LIN {X -0.031,Y -138.979,Z 1081.101,A 0.000,B 0.000,C 90.000,E1 198.181} C_DIS
LIN {X -0.046,Y -138.332,Z 1081.054,A 0.000,B 0.000,C 90.000,E1 189.782} C_DIS
LIN {X -0.046,Y -139.429,Z 1081.008,A 0.000,B 0.000,C 90.000,E1 181.375} C_DIS
LIN {X 0.007,Y -141.357,Z 1080.971,A 0.000,B 0.000,C 90.000,E1 174.837} C_DIS
LIN {X -0.016,Y -142.711,Z 1080.956,A 0.000,B 0.000,C 90.000,E1 172.064} C_DIS
LIN {X -0.057,Y -145.086,Z 1080.930,A 0.000,B 0.000,C 90.000,E1 167.465} C_DIS
LIN {X -0.062,Y -147.710,Z 1080.910,A 0.000,B 0.000,C 90.000,E1 163.795} C_DIS
LIN {X 0.022,Y -150.365,Z 1080.890,A 0.000,B 0.000,C 90.000,E1 160.115} C_DIS
LIN {X 0.040,Y -153.792,Z 1080.870,A 0.000,B 0.000,C 90.000,E1 156.485} C_DIS
LIN {X -0.040,Y -157.204,Z 1080.849,A 0.000,B 0.000,C 90.000,E1 152.922} C_DIS
LIN {X 0.041,Y -161.367,Z 1080.830,A 0.000,B 0.000,C 90.000,E1 149.331} C_DIS
LIN {X 0.053,Y -165.569,Z 1080.810,A 0.000,B 0.000,C 90.000,E1 145.801} C_DIS
LIN {X -0.064,Y -170.487,Z 1080.791,A 0.000,B 0.000,C 90.000,E1 142.351} C_DIS
LIN {X 0.086,Y -175.368,Z 1080.772,A 0.000,B 0.000,C 90.000,E1 138.852} C_DIS
LIN {X -0.052,Y -180.992,Z 1080.753,A 0.000,B 0.000,C 90.000,E1 135.486} C_DIS
LIN {X 0.073,Y -186.419,Z 1080.734,A 0.000,B 0.000,C 90.000,E1 132.081} C_DIS
LIN {X -0.127,Y -191.046,Z 1080.720,A 0.000,B 0.000,C 90.000,E1 129.644} C_DIS
LIN {X 0.065,Y -196.830,Z 1080.702,A 0.000,B 0.000,C 90.000,E1 126.297} C_DIS
LIN {X -0.010,Y -199.393,Z 1080.695,A 0.000,B 0.000,C 90.000,E1 125.025} C_DIS
LIN {X -0.069,Y -306.720,Z 1080.694,A 0.000,B 0.000,C 90.000,E1 125.025} C_DIS
LIN {X 0.023,Y -308.438,Z 1080.694,A 0.000,B 0.000,C 90.000,E1 124.978} C_DIS
LIN {X -0.026,Y -314.042,Z 1080.693,A 0.000,B 0.000,C 90.000,E1 124.692} C_DIS
LIN {X 0.025,Y -317.211,Z 1080.691,A 0.000,B 0.000,C 90.000,E1 124.358} C_DIS
LIN {X 0.033,Y -319.218,Z 1080.689,A 0.000,B 0.000,C 90.000,E1 124.072} C_DIS
LIN {X 0.038,Y -320.797,Z 1080.688,A 0.000,B 0.000,C 90.000,E1 123.785} C_DIS
LIN {X -0.151,Y -322.205,Z 1080.686,A 0.000,B 0.000,C 90.000,E1 123.499} C_DIS
LIN {X -0.148,Y -333.797,Z 1080.668,A 0.000,B 0.000,C 90.000,E1 120.335} C_DIS
LIN {X 0.027,Y -345.608,Z 1080.653,A 0.000,B 0.000,C 90.000,E1 117.513} C_DIS
LIN {X 0.075,Y -358.869,Z 1080.638,A 0.000,B 0.000,C 90.000,E1 114.771} C_DIS
LIN {X 0.107,Y -371.973,Z 1080.625,A 0.000,B 0.000,C 90.000,E1 112.386} C_DIS
LIN {X 0.047,Y -386.409,Z 1080.612,A 0.000,B 0.000,C 90.000,E1 110.066} C_DIS
LIN {X -0.152,Y -402.280,Z 1080.599,A 0.000,B 0.000,C 90.000,E1 107.819} C_DIS
LIN {X -0.217,Y -419.698,Z 1080.587,A 0.000,B 0.000,C 90.000,E1 105.607} C_DIS
LIN {X 0.053,Y -438.766,Z 1080.575,A 0.000,B 0.000,C 90.000,E1 103.411} C_DIS
LIN {X -0.227,Y -458.853,Z 1080.563,A 0.000,B 0.000,C 90.000,E1 101.422} C_DIS
LIN {X 0.154,Y -466.543,Z 1080.559,A 0.000,B 0.000,C 90.000,E1 100.658} C_DIS
LIN {X 0.100,Y -468.893,Z 1080.558,A 0.000,B 0.000,C 90.000,E1 100.433} C_DIS
LIN {X 0.129,Y -470.675,Z 1080.557,A 0.000,B 0.000,C 90.000,E1 100.197} C_DIS
LIN {X -0.017,Y -472.152,Z 1080.555,A 0.000,B 0.000,C 90.000,E1 99.962} C_DIS
LIN {X -0.166,Y -473.255,Z 1080.554,A 0.000,B 0.000,C 90.000,E1 99.726} C_DIS
LIN {X -0.057,Y -474.562,Z 1080.551,A 0.000,B 0.000,C 90.000,E1 99.208} C_DIS
LIN {X 0.134,Y -474.854,Z 1080.548,A 0.000,B 0.000,C 90.000,E1 98.681} C_DIS
LIN {X -0.211,Y -474.182,Z 1080.546,A 0.000,B 0.000,C 90.000,E1 98.219} C_DIS
LIN {X -0.081,Y -472.439,Z 1080.543,A 0.000,B 0.000,C 90.000,E1 97.701} C_DIS
LIN {X 0.246,Y -471.068,Z 1080.541,A 0.000,B 0.000,C 90.000,E1 97.409} C_DIS
LIN {X 0.119,Y -456.819,Z 1080.530,A 0.000,B 0.000,C 90.000,E1 95.391} C_DIS
LIN {X -0.179,Y -440.793,Z 1080.517,A 0.000,B 0.000,C 90.000,E1 93.094} C_DIS
LIN {X -0.040,Y -426.238,Z 1080.504,A 0.000,B 0.000,C 90.000,E1 90.688} C_DIS
LIN {X 0.135,Y -412.442,Z 1080.490,A 0.000,B 0.000,C 90.000,E1 88.224} C_DIS
LIN {X -0.194,Y -403.581,Z 1080.481,A 0.000,B 0.000,C 90.000,E1 86.617} C_DIS
LIN {X 0.099,Y -396.041,Z 1080.473,A 0.000,B 0.000,C 90.000,E1 85.179} C_DIS
LIN {X -0.069,Y -385.270,Z 1080.462,A 0.000,B 0.000,C 90.000,E1 83.223} C_DIS
LIN {X -0.004,Y -375.970,Z 1080.453,A 0.000,B 0.000,C 90.000,E1 81.489} C_DIS
LIN {X -0.045,Y -367.960,Z 1080.445,A 0.000,B 0.000,C 90.000,E1 80.038} C_DIS
LIN {X -0.168,Y -358.125,Z 1080.435,A 0.000,B 0.000,C 90.000,E1 78.285} C_DIS
LIN {X -0.044,Y -348.134,Z 1080.425,A 0.000,B 0.000,C 90.000,E1 76.464} C_DIS
LIN {X 0.188,Y -334.929,Z 1080.411,A 0.000,B 0.000,C 90.000,E1 73.976} C_DIS
LIN {X -0.184,Y -320.619,Z 1080.396,A 0.000,B 0.000,C 90.000,E1 71.221} C_DIS
LIN {X -0.014,Y -305.773,Z 1080.378,A 0.000,B 0.000,C 90.000,E1 67.975} C_DIS
LIN {X -0.091,Y -294.365,Z 1080.363,A 0.000,B 0.000,C 90.000,E1 65.357} C_DIS
LIN {X -0.072,Y -283.185,Z 1080.348,A 0.000,B 0.000,C 90.000,E1 62.666} C_DIS
LIN {X -0.064,Y -272.260,Z 1080.333,A 0.000,B 0.000,C 90.000,E1 59.921} C_DIS
LIN {X -0.013,Y -260.423,Z 1080.315,A 0.000,B 0.000,C 90.000,E1 56.755} C_DIS
LIN {X -0.074,Y -249.075,Z 1080.297,A 0.000,B 0.000,C 90.000,E1 53.543} C_DIS
LIN {X -0.021,Y -238.335,Z 1080.279,A 0.000,B 0.000,C 90.000,E1 50.231} C_DIS
LIN {X -0.028,Y -228.308,Z 1080.260,A 0.000,B 0.000,C 90.000,E1 46.863} C_DIS
LIN {X 0.095,Y -219.962,Z 1080.243,A 0.000,B 0.000,C 90.000,E1 43.785} C_DIS
LIN {X 0.030,Y -211.982,Z 1080.226,A 0.000,B 0.000,C 90.000,E1 40.701} C_DIS
LIN {X -0.048,Y -204.413,Z 1080.209,A 0.000,B 0.000,C 90.000,E1 37.569} C_DIS
LIN {X 0.085,Y -197.482,Z 1080.191,A 0.000,B 0.000,C 90.000,E1 34.326} C_DIS
LIN {X 0.049,Y -191.144,Z 1080.173,A 0.000,B 0.000,C 90.000,E1 31.082} C_DIS
LIN {X 0.090,Y -185.554,Z 1080.154,A 0.000,B 0.000,C 90.000,E1 27.769} C_DIS
LIN {X -0.022,Y -180.742,Z 1080.136,A 0.000,B 0.000,C 90.000,E1 24.463} C_DIS
LIN {X -0.063,Y -176.577,Z 1080.117,A 0.000,B 0.000,C 90.000,E1 21.099} C_DIS
LIN {X -0.069,Y -173.092,Z 1080.098,A 0.000,B 0.000,C 90.000,E1 17.692} C_DIS
LIN {X 0.045,Y -169.742,Z 1080.074,A 0.000,B 0.000,C 90.000,E1 13.355} C_DIS
LIN {X 0.023,Y -167.058,Z 1080.045,A 0.000,B 0.000,C 90.000,E1 8.163} C_DIS
LIN {X 0.051,Y -167.588,Z 1079.954,A 0.000,B 0.000,C 90.000,E1 351.659} C_DIS
LIN {X -0.059,Y -170.073,Z 1079.930,A 0.000,B 0.000,C 90.000,E1 347.353} C_DIS
LIN {X 0.007,Y -173.624,Z 1079.906,A 0.000,B 0.000,C 90.000,E1 343.015} C_DIS
LIN {X 0.062,Y -178.236,Z 1079.882,A 0.000,B 0.000,C 90.000,E1 338.720} C_DIS
LIN {X -0.018,Y -182.666,Z 1079.863,A 0.000,B 0.000,C 90.000,E1 335.357} C_DIS
LIN {X 0.076,Y -187.791,Z 1079.844,A 0.000,B 0.000,C 90.000,E1 331.975} C_DIS
LIN {X -0.097,Y -192.235,Z 1079.831,A 0.000,B 0.000,C 90.000,E1 329.537} C_DIS
LIN {X 0.048,Y -198.868,Z 1079.812,A 0.000,B 0.000,C 90.000,E1 326.215} C_DIS
LIN {X -0.027,Y -206.227,Z 1079.794,A 0.000,B 0.000,C 90.000,E1 323.004} C_DIS
LIN {X -0.128,Y -215.311,Z 1079.775,A 0.000,B 0.000,C 90.000,E1 319.461} C_DIS
LIN {X 0.000,Y -225.348,Z 1079.755,A 0.000,B 0.000,C 90.000,E1 315.931} C_DIS
LIN {X -0.025,Y -235.355,Z 1079.738,A 0.000,B 0.000,C 90.000,E1 312.894} C_DIS
LIN {X 0.113,Y -243.794,Z 1079.726,A 0.000,B 0.000,C 90.000,E1 310.620} C_DIS
LIN {X -0.065,Y -254.986,Z 1079.712,A 0.000,B 0.000,C 90.000,E1 308.096} C_DIS
LIN {X -0.011,Y -265.577,Z 1079.700,A 0.000,B 0.000,C 90.000,E1 305.931} C_DIS
LIN {X 0.140,Y -282.884,Z 1079.682,A 0.000,B 0.000,C 90.000,E1 302.752} C_DIS
LIN {X -0.038,Y -301.712,Z 1079.665,A 0.000,B 0.000,C 90.000,E1 299.745} C_DIS
LIN {X -0.051,Y -319.749,Z 1079.651,A 0.000,B 0.000,C 90.000,E1 297.129} C_DIS
LIN {X 0.005,Y -331.675,Z 1079.642,A 0.000,B 0.000,C 90.000,E1 295.540} C_DIS
LIN {X -0.092,Y -344.652,Z 1079.633,A 0.000,B 0.000,C 90.000,E1 294.003} C_DIS
LIN {X -0.034,Y -360.721,Z 1079.624,A 0.000,B 0.000,C 90.000,E1 292.280} C_DIS
LIN {X 0.134,Y -379.510,Z 1079.614,A 0.000,B 0.000,C 90.000,E1 290.482} C_DIS
LIN {X -0.097,Y -398.773,Z 1079.605,A 0.000,B 0.000,C 90.000,E1 288.852} C_DIS
LIN {X -0.116,Y -409.487,Z 1079.599,A 0.000,B 0.000,C 90.000,E1 287.928} C_DIS
LIN {X -0.081,Y -419.968,Z 1079.594,A 0.000,B 0.000,C 90.000,E1 286.985} C_DIS
LIN {X -0.117,Y -427.580,Z 1079.590,A 0.000,B 0.000,C 90.000,E1 286.260} C_DIS
LIN {X -0.015,Y -435.113,Z 1079.586,A 0.000,B 0.000,C 90.000,E1 285.481} C_DIS
LIN {X -0.191,Y -442.406,Z 1079.582,A 0.000,B 0.000,C 90.000,E1 284.717} C_DIS
LIN {X 0.146,Y -449.233,Z 1079.577,A 0.000,B 0.000,C 90.000,E1 283.883} C_DIS
LIN {X -0.005,Y -455.567,Z 1079.573,A 0.000,B 0.000,C 90.000,E1 283.119} C_DIS
LIN {X -0.097,Y -461.188,Z 1079.569,A 0.000,B 0.000,C 90.000,E1 282.355} C_DIS
LIN {X -0.149,Y -466.074,Z 1079.564,A 0.000,B 0.000,C 90.000,E1 281.591} C_DIS
LIN {X -0.243,Y -470.161,Z 1079.560,A 0.000,B 0.000,C 90.000,E1 280.838} C_DIS
LIN {X 0.248,Y -473.587,Z 1079.556,A 0.000,B 0.000,C 90.000,E1 280.018} C_DIS
LIN {X -0.110,Y -475.562,Z 1079.553,A 0.000,B 0.000,C 90.000,E1 279.557} C_DIS
LIN {X 0.086,Y -477.292,Z 1079.550,A 0.000,B 0.000,C 90.000,E1 279.029} C_DIS
LIN {X -0.112,Y -480.068,Z 1079.545,A 0.000,B 0.000,C 90.000,E1 278.049} C_DIS
LIN {X 0.208,Y -482.037,Z 1079.539,A 0.000,B 0.000,C 90.000,E1 277.011} C_DIS
LIN {X -0.099,Y -482.717,Z 1079.536,A 0.000,B 0.000,C 90.000,E1 276.549} C_DIS
LIN {X 0.078,Y -483.184,Z 1079.534,A 0.000,B 0.000,C 90.000,E1 276.030} C_DIS
LIN {X -0.223,Y -483.240,Z 1079.531,A 0.000,B 0.000,C 90.000,E1 275.568} C_DIS
LIN {X -0.040,Y -482.989,Z 1079.528,A 0.000,B 0.000,C 90.000,E1 275.049} C_DIS
LIN {X 0.139,Y -482.213,Z 1079.525,A 0.000,B 0.000,C 90.000,E1 274.531} C_DIS
LIN {X -0.165,Y -480.947,Z 1079.522,A 0.000,B 0.000,C 90.000,E1 274.069} C_DIS
LIN {X -0.026,Y -479.128,Z 1079.520,A 0.000,B 0.000,C 90.000,E1 273.555} C_DIS
LIN {X 0.134,Y -476.657,Z 1079.517,A 0.000,B 0.000,C 90.000,E1 273.037} C_DIS
LIN {X -0.223,Y -473.411,Z 1079.514,A 0.000,B 0.000,C 90.000,E1 272.579} C_DIS
LIN {X -0.119,Y -469.277,Z 1079.511,A 0.000,B 0.000,C 90.000,E1 272.064} C_DIS
LIN {X -0.021,Y -464.125,Z 1079.509,A 0.000,B 0.000,C 90.000,E1 271.547} C_DIS
LIN {X -0.149,Y -458.207,Z 1079.506,A 0.000,B 0.000,C 90.000,E1 271.088} C_DIS
LIN {X 0.162,Y -451.915,Z 1079.504,A 0.000,B 0.000,C 90.000,E1 270.630} C_DIS
LIN {X 0.015,Y -445.005,Z 1079.502,A 0.000,B 0.000,C 90.000,E1 270.286} C_DIS
LIN {X -0.052,Y -437.619,Z 1079.500,A 0.000,B 0.000,C 90.000,E1 270.000} C_DIS
LIN {X -0.035,Y -430.037,Z 1079.499,A 0.000,B 0.000,C 90.000,E1 269.771} C_DIS
LIN {X -0.036,Y -422.471,Z 1079.498,A 0.000,B 0.000,C 90.000,E1 269.599} C_DIS
LIN {X -0.167,Y -414.182,Z 1079.497,A 0.000,B 0.000,C 90.000,E1 269.484} C_DIS
LIN {X -0.071,Y -404.523,Z 1079.496,A 0.000,B 0.000,C 90.000,E1 269.370} C_DIS
LIN {X 0.006,Y -396.170,Z 1079.496,A 0.000,B 0.000,C 90.000,E1 269.312} C_DIS
LIN {X -0.059,Y -391.384,Z 1079.496,A 0.000,B 0.000,C 90.000,E1 269.312} C_DIS
LIN {X -0.057,Y -181.388,Z 1079.496,A 0.000,B 0.000,C 90.000,E1 269.312} C_DIS
LIN {X 0.061,Y -180.784,Z 1079.471,A 0.000,B 0.000,C 90.000,E1 264.723} C_DIS
LIN {X -0.045,Y -178.881,Z 1079.443,A 0.000,B 0.000,C 90.000,E1 259.690} C_DIS
LIN {X 0.032,Y -175.923,Z 1079.414,A 0.000,B 0.000,C 90.000,E1 254.574} C_DIS
LIN {X -0.023,Y -175.361,Z 1079.410,A 0.000,B 0.000,C 90.000,E1 253.740} C_DIS
LIN {X 0.036,Y -172.140,Z 1079.386,A 0.000,B 0.000,C 90.000,E1 249.444} C_DIS
LIN {X 0.013,Y -171.604,Z 1079.381,A 0.000,B 0.000,C 90.000,E1 248.592} C_DIS
LIN {X 0.002,Y -167.826,Z 1079.357,A 0.000,B 0.000,C 90.000,E1 244.280} C_DIS
LIN {X 0.019,Y -166.551,Z 1079.347,A 0.000,B 0.000,C 90.000,E1 242.538} C_DIS
LIN {X -0.070,Y -162.547,Z 1079.323,A 0.000,B 0.000,C 90.000,E1 238.201} C_DIS
LIN {X -0.010,Y -161.224,Z 1079.313,A 0.000,B 0.000,C 90.000,E1 236.421} C_DIS
LIN {X 0.025,Y -157.230,Z 1079.289,A 0.000,B 0.000,C 90.000,E1 231.984} C_DIS
LIN {X 0.048,Y -155.956,Z 1079.279,A 0.000,B 0.000,C 90.000,E1 230.194} C_DIS
LIN {X 0.006,Y -152.209,Z 1079.254,A 0.000,B 0.000,C 90.000,E1 225.729} C_DIS
LIN {X 0.028,Y -150.454,Z 1079.239,A 0.000,B 0.000,C 90.000,E1 223.014} C_DIS
LIN {X 0.054,Y -147.180,Z 1079.214,A 0.000,B 0.000,C 90.000,E1 218.463} C_DIS
LIN {X 0.020,Y -145.196,Z 1079.193,A 0.000,B 0.000,C 90.000,E1 214.818} C_DIS
LIN {X 0.054,Y -142.336,Z 1079.163,A 0.000,B 0.000,C 90.000,E1 209.283} C_DIS
LIN {X -0.016,Y -141.725,Z 1079.153,A 0.000,B 0.000,C 90.000,E1 207.462} C_DIS
LIN {X -0.034,Y -139.478,Z 1079.116,A 0.000,B 0.000,C 90.000,E1 200.972} C_DIS
LIN {X -0.045,Y -138.978,Z 1079.101,A 0.000,B 0.000,C 90.000,E1 198.181} C_DIS
LIN {X 0.076,Y -138.332,Z 1079.054,A 0.000,B 0.000,C 90.000,E1 189.726} C_DIS
LIN {X -0.059,Y -139.431,Z 1079.007,A 0.000,B 0.000,C 90.000,E1 181.375} C_DIS
LIN {X 0.020,Y -140.956,Z 1078.976,A 0.000,B 0.000,C 90.000,E1 175.755} C_DIS
LIN {X -0.030,Y -142.713,Z 1078.956,A 0.000,B 0.000,C 90.000,E1 172.064} C_DIS
LIN {X 0.070,Y -145.089,Z 1078.930,A 0.000,B 0.000,C 90.000,E1 167.409} C_DIS
LIN {X 0.065,Y -147.713,Z 1078.910,A 0.000,B 0.000,C 90.000,E1 163.740} C_DIS
LIN {X 0.007,Y -150.370,Z 1078.890,A 0.000,B 0.000,C 90.000,E1 160.115} C_DIS
LIN {X 0.025,Y -153.798,Z 1078.869,A 0.000,B 0.000,C 90.000,E1 156.485} C_DIS
LIN {X 0.085,Y -157.210,Z 1078.849,A 0.000,B 0.000,C 90.000,E1 152.871} C_DIS
LIN {X 0.026,Y -161.373,Z 1078.830,A 0.000,B 0.000,C 90.000,E1 149.331} C_DIS
LIN {X 0.038,Y -165.576,Z 1078.810,A 0.000,B 0.000,C 90.000,E1 145.801} C_DIS
LIN {X 0.024,Y -170.496,Z 1078.791,A 0.000,B 0.000,C 90.000,E1 142.316} C_DIS
LIN {X 0.069,Y -175.376,Z 1078.771,A 0.000,B 0.000,C 90.000,E1 138.852} C_DIS
LIN {X -0.068,Y -181.000,Z 1078.753,A 0.000,B 0.000,C 90.000,E1 135.486} C_DIS
LIN {X 0.056,Y -186.428,Z 1078.734,A 0.000,B 0.000,C 90.000,E1 132.081} C_DIS
LIN {X 0.125,Y -191.054,Z 1078.720,A 0.000,B 0.000,C 90.000,E1 129.564} C_DIS
LIN {X 0.048,Y -196.839,Z 1078.702,A 0.000,B 0.000,C 90.000,E1 126.297} C_DIS
LIN {X 0.133,Y -199.309,Z 1078.695,A 0.000,B 0.000,C 90.000,E1 125.025} C_DIS
LIN {X 0.145,Y -306.793,Z 1078.695,A 0.000,B 0.000,C 90.000,E1 125.025} C_DIS
LIN {X -0.037,Y -308.518,Z 1078.695,A 0.000,B 0.000,C 90.000,E1 125.025} C_DIS
LIN {X 0.172,Y -312.221,Z 1078.694,A 0.000,B 0.000,C 90.000,E1 124.818} C_DIS
LIN {X -0.053,Y -314.434,Z 1078.693,A 0.000,B 0.000,C 90.000,E1 124.692} C_DIS
LIN {X -0.074,Y -318.322,Z 1078.690,A 0.000,B 0.000,C 90.000,E1 124.246} C_DIS
LIN {X 0.049,Y -320.192,Z 1078.688,A 0.000,B 0.000,C 90.000,E1 123.913} C_DIS
LIN {X -0.094,Y -321.659,Z 1078.687,A 0.000,B 0.000,C 90.000,E1 123.627} C_DIS
LIN {X 0.140,Y -335.736,Z 1078.666,A 0.000,B 0.000,C 90.000,E1 119.795} C_DIS
LIN {X -0.090,Y -347.789,Z 1078.650,A 0.000,B 0.000,C 90.000,E1 117.052} C_DIS
LIN {X -0.146,Y -361.319,Z 1078.635,A 0.000,B 0.000,C 90.000,E1 114.335} C_DIS
LIN {X -0.060,Y -374.676,Z 1078.622,A 0.000,B 0.000,C 90.000,E1 111.950} C_DIS
LIN {X -0.061,Y -389.386,Z 1078.609,A 0.000,B 0.000,C 90.000,E1 109.631} C_DIS
LIN {X 0.065,Y -405.552,Z 1078.596,A 0.000,B 0.000,C 90.000,E1 107.347} C_DIS
LIN {X 0.097,Y -423.289,Z 1078.584,A 0.000,B 0.000,C 90.000,E1 105.134} C_DIS
LIN {X -0.023,Y -442.658,Z 1078.572,A 0.000,B 0.000,C 90.000,E1 103.008} C_DIS
LIN {X 0.062,Y -462.856,Z 1078.561,A 0.000,B 0.000,C 90.000,E1 101.007} C_DIS
LIN {X -0.023,Y -467.950,Z 1078.559,A 0.000,B 0.000,C 90.000,E1 100.546} C_DIS
LIN {X -0.030,Y -469.985,Z 1078.557,A 0.000,B 0.000,C 90.000,E1 100.310} C_DIS
LIN {X -0.038,Y -471.530,Z 1078.556,A 0.000,B 0.000,C 90.000,E1 100.074} C_DIS
LIN {X 0.201,Y -472.784,Z 1078.555,A 0.000,B 0.000,C 90.000,E1 99.792} C_DIS
LIN {X 0.056,Y -473.704,Z 1078.553,A 0.000,B 0.000,C 90.000,E1 99.557} C_DIS
LIN {X 0.246,Y -474.711,Z 1078.550,A 0.000,B 0.000,C 90.000,E1 99.029} C_DIS
LIN {X -0.103,Y -474.732,Z 1078.547,A 0.000,B 0.000,C 90.000,E1 98.568} C_DIS
LIN {X 0.025,Y -473.777,Z 1078.545,A 0.000,B 0.000,C 90.000,E1 98.049} C_DIS
LIN {X 0.154,Y -471.684,Z 1078.542,A 0.000,B 0.000,C 90.000,E1 97.530} C_DIS
LIN {X -0.187,Y -468.228,Z 1078.539,A 0.000,B 0.000,C 90.000,E1 97.068} C_DIS
LIN {X -0.124,Y -455.799,Z 1078.529,A 0.000,B 0.000,C 90.000,E1 95.277} C_DIS
LIN {X -0.205,Y -441.518,Z 1078.518,A 0.000,B 0.000,C 90.000,E1 93.212} C_DIS
LIN {X 0.113,Y -425.345,Z 1078.503,A 0.000,B 0.000,C 90.000,E1 90.516} C_DIS
LIN {X 0.028,Y -408.666,Z 1078.486,A 0.000,B 0.000,C 90.000,E1 87.535} C_DIS
LIN {X 0.044,Y -399.759,Z 1078.477,A 0.000,B 0.000,C 90.000,E1 85.869} C_DIS
LIN {X -0.048,Y -389.033,Z 1078.466,A 0.000,B 0.000,C 90.000,E1 83.913} C_DIS
LIN {X 0.063,Y -378.216,Z 1078.455,A 0.000,B 0.000,C 90.000,E1 81.894} C_DIS
LIN {X 0.053,Y -368.646,Z 1078.445,A 0.000,B 0.000,C 90.000,E1 80.151} C_DIS
LIN {X -0.129,Y -358.801,Z 1078.436,A 0.000,B 0.000,C 90.000,E1 78.409} C_DIS
LIN {X 0.002,Y -348.832,Z 1078.426,A 0.000,B 0.000,C 90.000,E1 76.589} C_DIS
LIN {X 0.018,Y -337.247,Z 1078.414,A 0.000,B 0.000,C 90.000,E1 74.448} C_DIS
LIN {X 0.027,Y -322.815,Z 1078.398,A 0.000,B 0.000,C 90.000,E1 71.638} C_DIS
LIN {X -0.139,Y -307.817,Z 1078.380,A 0.000,B 0.000,C 90.000,E1 68.465} C_DIS
LIN {X 0.114,Y -296.351,Z 1078.366,A 0.000,B 0.000,C 90.000,E1 65.793} C_DIS
LIN {X 0.069,Y -286.517,Z 1078.353,A 0.000,B 0.000,C 90.000,E1 63.461} C_DIS
LIN {X 0.145,Y -275.497,Z 1078.338,A 0.000,B 0.000,C 90.000,E1 60.717} C_DIS
LIN {X -0.143,Y -264.801,Z 1078.322,A 0.000,B 0.000,C 90.000,E1 57.995} C_DIS
LIN {X 0.094,Y -254.490,Z 1078.306,A 0.000,B 0.000,C 90.000,E1 55.102} C_DIS
LIN {X 0.148,Y -244.623,Z 1078.290,A 0.000,B 0.000,C 90.000,E1 52.190} C_DIS
LIN {X -0.145,Y -234.131,Z 1078.272,A 0.000,B 0.000,C 90.000,E1 48.933} C_DIS
LIN {X -0.041,Y -225.430,Z 1078.255,A 0.000,B 0.000,C 90.000,E1 45.891} C_DIS
LIN {X 0.010,Y -217.158,Z 1078.238,A 0.000,B 0.000,C 90.000,E1 42.813} C_DIS
LIN {X -0.103,Y -209.272,Z 1078.221,A 0.000,B 0.000,C 90.000,E1 39.725} C_DIS
LIN {X 0.075,Y -201.926,Z 1078.203,A 0.000,B 0.000,C 90.000,E1 36.503} C_DIS
LIN {X 0.032,Y -195.149,Z 1078.185,A 0.000,B 0.000,C 90.000,E1 33.293} C_DIS
LIN {X 0.102,Y -189.040,Z 1078.167,A 0.000,B 0.000,C 90.000,E1 30.001} C_DIS
LIN {X -0.089,Y -183.713,Z 1078.148,A 0.000,B 0.000,C 90.000,E1 26.744} C_DIS
LIN {X -0.078,Y -179.114,Z 1078.130,A 0.000,B 0.000,C 90.000,E1 23.387} C_DIS
LIN {X -0.063,Y -175.159,Z 1078.111,A 0.000,B 0.000,C 90.000,E1 19.993} C_DIS
LIN {X 0.002,Y -171.899,Z 1078.092,A 0.000,B 0.000,C 90.000,E1 16.551} C_DIS
LIN {X -0.005,Y -168.836,Z 1078.068,A 0.000,B 0.000,C 90.000,E1 12.243} C_DIS
LIN {X 0.046,Y -166.198,Z 1078.034,A 0.000,B 0.000,C 90.000,E1 6.144} C_DIS
LIN {X 0.029,Y -167.013,Z 1077.959,A 0.000,B 0.000,C 90.000,E1 352.534} C_DIS
LIN {X -0.077,Y -169.876,Z 1077.930,A 0.000,B 0.000,C 90.000,E1 347.353} C_DIS
LIN {X -0.016,Y -173.445,Z 1077.906,A 0.000,B 0.000,C 90.000,E1 343.015} C_DIS
LIN {X 0.034,Y -177.040,Z 1077.887,A 0.000,B 0.000,C 90.000,E1 339.571} C_DIS
LIN {X 0.024,Y -181.331,Z 1077.868,A 0.000,B 0.000,C 90.000,E1 336.177} C_DIS
LIN {X 0.001,Y -186.257,Z 1077.849,A 0.000,B 0.000,C 90.000,E1 332.820} C_DIS
LIN {X -0.035,Y -190.532,Z 1077.835,A 0.000,B 0.000,C 90.000,E1 330.333} C_DIS
LIN {X -0.038,Y -196.978,Z 1077.817,A 0.000,B 0.000,C 90.000,E1 327.041} C_DIS
LIN {X 0.005,Y -204.202,Z 1077.799,A 0.000,B 0.000,C 90.000,E1 323.783} C_DIS
LIN {X -0.019,Y -212.093,Z 1077.781,A 0.000,B 0.000,C 90.000,E1 320.598} C_DIS
LIN {X -0.044,Y -220.675,Z 1077.764,A 0.000,B 0.000,C 90.000,E1 317.472} C_DIS
LIN {X 0.138,Y -230.094,Z 1077.747,A 0.000,B 0.000,C 90.000,E1 314.352} C_DIS
LIN {X -0.044,Y -239.333,Z 1077.732,A 0.000,B 0.000,C 90.000,E1 311.757} C_DIS
LIN {X 0.020,Y -248.271,Z 1077.720,A 0.000,B 0.000,C 90.000,E1 309.519} C_DIS
LIN {X -0.095,Y -258.244,Z 1077.707,A 0.000,B 0.000,C 90.000,E1 307.363} C_DIS
LIN {X 0.066,Y -273.015,Z 1077.692,A 0.000,B 0.000,C 90.000,E1 304.485} C_DIS
LIN {X 0.052,Y -291.007,Z 1077.674,A 0.000,B 0.000,C 90.000,E1 301.386} C_DIS
LIN {X -0.089,Y -308.291,Z 1077.660,A 0.000,B 0.000,C 90.000,E1 298.743} C_DIS
LIN {X -0.102,Y -329.252,Z 1077.644,A 0.000,B 0.000,C 90.000,E1 295.848} C_DIS
LIN {X 0.056,Y -342.075,Z 1077.635,A 0.000,B 0.000,C 90.000,E1 294.259} C_DIS
LIN {X 0.042,Y -355.244,Z 1077.627,A 0.000,B 0.000,C 90.000,E1 292.823} C_DIS
LIN {X -0.032,Y -374.367,Z 1077.616,A 0.000,B 0.000,C 90.000,E1 290.972} C_DIS
LIN {X 0.012,Y -393.690,Z 1077.607,A 0.000,B 0.000,C 90.000,E1 289.268} C_DIS
LIN {X -0.117,Y -407.467,Z 1077.600,A 0.000,B 0.000,C 90.000,E1 288.109} C_DIS
LIN {X 0.005,Y -418.077,Z 1077.595,A 0.000,B 0.000,C 90.000,E1 287.149} C_DIS
LIN {X -0.125,Y -425.791,Z 1077.591,A 0.000,B 0.000,C 90.000,E1 286.441} C_DIS
LIN {X 0.085,Y -433.260,Z 1077.587,A 0.000,B 0.000,C 90.000,E1 285.662} C_DIS
LIN {X 0.000,Y -440.537,Z 1077.583,A 0.000,B 0.000,C 90.000,E1 284.898} C_DIS
LIN {X -0.049,Y -447.485,Z 1077.578,A 0.000,B 0.000,C 90.000,E1 284.120} C_DIS
LIN {X -0.171,Y -453.916,Z 1077.574,A 0.000,B 0.000,C 90.000,E1 283.355} C_DIS
LIN {X 0.165,Y -459.735,Z 1077.570,A 0.000,B 0.000,C 90.000,E1 282.535} C_DIS
LIN {X 0.112,Y -464.865,Z 1077.565,A 0.000,B 0.000,C 90.000,E1 281.771} C_DIS
LIN {X 0.094,Y -469.138,Z 1077.561,A 0.000,B 0.000,C 90.000,E1 281.007} C_DIS
LIN {X 0.031,Y -472.754,Z 1077.557,A 0.000,B 0.000,C 90.000,E1 280.254} C_DIS
LIN {X -0.001,Y -475.834,Z 1077.553,A 0.000,B 0.000,C 90.000,E1 279.500} C_DIS
LIN {X 0.196,Y -477.551,Z 1077.550,A 0.000,B 0.000,C 90.000,E1 278.973} C_DIS
LIN {X -0.142,Y -479.042,Z 1077.547,A 0.000,B 0.000,C 90.000,E1 278.511} C_DIS
LIN {X 0.004,Y -480.332,Z 1077.544,A 0.000,B 0.000,C 90.000,E1 277.992} C_DIS
LIN {X -0.091,Y -482.325,Z 1077.539,A 0.000,B 0.000,C 90.000,E1 277.004} C_DIS
LIN {X 0.078,Y -483.018,Z 1077.536,A 0.000,B 0.000,C 90.000,E1 276.486} C_DIS
LIN {X 0.254,Y -483.442,Z 1077.533,A 0.000,B 0.000,C 90.000,E1 275.967} C_DIS
LIN {X -0.096,Y -483.538,Z 1077.531,A 0.000,B 0.000,C 90.000,E1 275.511} C_DIS
LIN {X 0.088,Y -483.223,Z 1077.528,A 0.000,B 0.000,C 90.000,E1 274.992} C_DIS
LIN {X -0.211,Y -482.431,Z 1077.525,A 0.000,B 0.000,C 90.000,E1 274.531} C_DIS
LIN {X -0.033,Y -481.125,Z 1077.522,A 0.000,B 0.000,C 90.000,E1 274.012} C_DIS
LIN {X 0.106,Y -479.277,Z 1077.520,A 0.000,B 0.000,C 90.000,E1 273.498} C_DIS
LIN {X -0.209,Y -476.758,Z 1077.517,A 0.000,B 0.000,C 90.000,E1 273.037} C_DIS
LIN {X -0.090,Y -473.440,Z 1077.514,A 0.000,B 0.000,C 90.000,E1 272.522} C_DIS
LIN {X 0.014,Y -469.253,Z 1077.511,A 0.000,B 0.000,C 90.000,E1 272.007} C_DIS
LIN {X -0.163,Y -466.788,Z 1077.510,A 0.000,B 0.000,C 90.000,E1 271.776} C_DIS
LIN {X 0.072,Y -461.196,Z 1077.507,A 0.000,B 0.000,C 90.000,E1 271.260} C_DIS
LIN {X 0.189,Y -455.133,Z 1077.505,A 0.000,B 0.000,C 90.000,E1 270.802} C_DIS
LIN {X -0.111,Y -451.816,Z 1077.503,A 0.000,B 0.000,C 90.000,E1 270.630} C_DIS
LIN {X 0.195,Y -444.754,Z 1077.501,A 0.000,B 0.000,C 90.000,E1 270.229} C_DIS
LIN {X -0.030,Y -441.441,Z 1077.501,A 0.000,B 0.000,C 90.000,E1 270.115} C_DIS
LIN {X 0.213,Y -434.099,Z 1077.499,A 0.000,B 0.000,C 90.000,E1 269.828} C_DIS
LIN {X 0.027,Y -426.617,Z 1077.498,A 0.000,B 0.000,C 90.000,E1 269.656} C_DIS
LIN {X 0.183,Y -418.588,Z 1077.497,A 0.000,B 0.000,C 90.000,E1 269.484} C_DIS
LIN {X 0.189,Y -409.875,Z 1077.497,A 0.000,B 0.000,C 90.000,E1 269.370} C_DIS
LIN {X -0.076,Y -396.410,Z 1077.496,A 0.000,B 0.000,C 90.000,E1 269.312} C_DIS
LIN {X -0.139,Y -391.628,Z 1077.496,A 0.000,B 0.000,C 90.000,E1 269.312} C_DIS
LIN {X 0.088,Y -181.384,Z 1077.496,A 0.000,B 0.000,C 90.000,E1 269.255} C_DIS
LIN {X 0.024,Y -180.779,Z 1077.471,A 0.000,B 0.000,C 90.000,E1 264.723} C_DIS
LIN {X -0.081,Y -178.876,Z 1077.443,A 0.000,B 0.000,C 90.000,E1 259.690} C_DIS
LIN {X -0.005,Y -175.919,Z 1077.414,A 0.000,B 0.000,C 90.000,E1 254.574} C_DIS
LIN {X 0.052,Y -174.614,Z 1077.405,A 0.000,B 0.000,C 90.000,E1 252.851} C_DIS
LIN {X -0.023,Y -171.594,Z 1077.381,A 0.000,B 0.000,C 90.000,E1 248.592} C_DIS
LIN {X -0.033,Y -167.817,Z 1077.357,A 0.000,B 0.000,C 90.000,E1 244.280} C_DIS
LIN {X -0.016,Y -166.540,Z 1077.347,A 0.000,B 0.000,C 90.000,E1 242.538} C_DIS
LIN {X -0.106,Y -162.537,Z 1077.323,A 0.000,B 0.000,C 90.000,E1 238.201} C_DIS
LIN {X -0.045,Y -161.213,Z 1077.313,A 0.000,B 0.000,C 90.000,E1 236.421} C_DIS
LIN {X -0.009,Y -157.221,Z 1077.289,A 0.000,B 0.000,C 90.000,E1 231.984} C_DIS
LIN {X 0.014,Y -155.947,Z 1077.279,A 0.000,B 0.000,C 90.000,E1 230.194} C_DIS
LIN {X -0.027,Y -152.200,Z 1077.254,A 0.000,B 0.000,C 90.000,E1 225.729} C_DIS
LIN {X -0.006,Y -150.446,Z 1077.239,A 0.000,B 0.000,C 90.000,E1 223.014} C_DIS
LIN {X 0.021,Y -147.172,Z 1077.214,A 0.000,B 0.000,C 90.000,E1 218.463} C_DIS
LIN {X -0.012,Y -145.188,Z 1077.193,A 0.000,B 0.000,C 90.000,E1 214.818} C_DIS
LIN {X 0.023,Y -142.331,Z 1077.163,A 0.000,B 0.000,C 90.000,E1 209.283} C_DIS
LIN {X -0.047,Y -141.720,Z 1077.152,A 0.000,B 0.000,C 90.000,E1 207.462} C_DIS
LIN {X 0.065,Y -139.476,Z 1077.116,A 0.000,B 0.000,C 90.000,E1 200.918} C_DIS
LIN {X -0.076,Y -138.974,Z 1077.101,A 0.000,B 0.000,C 90.000,E1 198.181} C_DIS
LIN {X 0.045,Y -138.331,Z 1077.054,A 0.000,B 0.000,C 90.000,E1 189.726} C_DIS
LIN {X 0.048,Y -139.434,Z 1077.007,A 0.000,B 0.000,C 90.000,E1 181.318} C_DIS
LIN {X -0.012,Y -140.962,Z 1076.976,A 0.000,B 0.000,C 90.000,E1 175.755} C_DIS
LIN {X -0.062,Y -142.717,Z 1076.956,A 0.000,B 0.000,C 90.000,E1 172.064} C_DIS
LIN {X 0.038,Y -145.097,Z 1076.930,A 0.000,B 0.000,C 90.000,E1 167.409} C_DIS
LIN {X 0.032,Y -147.722,Z 1076.910,A 0.000,B 0.000,C 90.000,E1 163.740} C_DIS
LIN {X -0.027,Y -150.380,Z 1076.890,A 0.000,B 0.000,C 90.000,E1 160.115} C_DIS
LIN {X -0.009,Y -153.811,Z 1076.869,A 0.000,B 0.000,C 90.000,E1 156.485} C_DIS
LIN {X 0.051,Y -157.223,Z 1076.849,A 0.000,B 0.000,C 90.000,E1 152.871} C_DIS
LIN {X -0.008,Y -161.389,Z 1076.830,A 0.000,B 0.000,C 90.000,E1 149.331} C_DIS
LIN {X 0.002,Y -165.591,Z 1076.810,A 0.000,B 0.000,C 90.000,E1 145.801} C_DIS
LIN {X -0.011,Y -170.514,Z 1076.791,A 0.000,B 0.000,C 90.000,E1 142.316} C_DIS
LIN {X 0.033,Y -175.394,Z 1076.771,A 0.000,B 0.000,C 90.000,E1 138.852} C_DIS
LIN {X -0.105,Y -181.018,Z 1076.753,A 0.000,B 0.000,C 90.000,E1 135.486} C_DIS
LIN {X 0.018,Y -186.448,Z 1076.734,A 0.000,B 0.000,C 90.000,E1 132.081} C_DIS
LIN {X 0.087,Y -191.074,Z 1076.720,A 0.000,B 0.000,C 90.000,E1 129.564} C_DIS
LIN {X 0.009,Y -196.861,Z 1076.702,A 0.000,B 0.000,C 90.000,E1 126.297} C_DIS
LIN {X 0.024,Y -199.211,Z 1076.695,A 0.000,B 0.000,C 90.000,E1 125.105} C_DIS
LIN {X -0.005,Y -305.919,Z 1076.695,A 0.000,B 0.000,C 90.000,E1 125.105} C_DIS
LIN {X -0.060,Y -312.160,Z 1076.694,A 0.000,B 0.000,C 90.000,E1 124.898} C_DIS
LIN {X -0.115,Y -314.857,Z 1076.693,A 0.000,B 0.000,C 90.000,E1 124.692} C_DIS
LIN {X 0.008,Y -318.653,Z 1076.690,A 0.000,B 0.000,C 90.000,E1 124.199} C_DIS
LIN {X 0.072,Y -320.467,Z 1076.688,A 0.000,B 0.000,C 90.000,E1 123.865} C_DIS
LIN {X -0.131,Y -321.883,Z 1076.686,A 0.000,B 0.000,C 90.000,E1 123.579} C_DIS
LIN {X -0.005,Y -334.672,Z 1076.667,A 0.000,B 0.000,C 90.000,E1 120.079} C_DIS
LIN {X -0.104,Y -346.597,Z 1076.652,A 0.000,B 0.000,C 90.000,E1 117.308} C_DIS
LIN {X -0.041,Y -359.983,Z 1076.636,A 0.000,B 0.000,C 90.000,E1 114.567} C_DIS
LIN {X -0.136,Y -373.205,Z 1076.623,A 0.000,B 0.000,C 90.000,E1 112.206} C_DIS
LIN {X -0.038,Y -387.768,Z 1076.610,A 0.000,B 0.000,C 90.000,E1 109.866} C_DIS
LIN {X 0.041,Y -403.777,Z 1076.598,A 0.000,B 0.000,C 90.000,E1 107.583} C_DIS
LIN {X 0.024,Y -421.344,Z 1076.585,A 0.000,B 0.000,C 90.000,E1 105.371} C_DIS
LIN {X -0.172,Y -440.562,Z 1076.573,A 0.000,B 0.000,C 90.000,E1 103.244} C_DIS
LIN {X 0.218,Y -460.702,Z 1076.562,A 0.000,B 0.000,C 90.000,E1 101.186} C_DIS
LIN {X 0.106,Y -468.312,Z 1076.558,A 0.000,B 0.000,C 90.000,E1 100.489} C_DIS
LIN {X 0.076,Y -470.269,Z 1076.557,A 0.000,B 0.000,C 90.000,E1 100.254} C_DIS
LIN {X 0.044,Y -471.755,Z 1076.556,A 0.000,B 0.000,C 90.000,E1 100.018} C_DIS
LIN {X -0.181,Y -472.942,Z 1076.554,A 0.000,B 0.000,C 90.000,E1 99.792} C_DIS
LIN {X 0.141,Y -473.807,Z 1076.553,A 0.000,B 0.000,C 90.000,E1 99.500} C_DIS
LIN {X -0.136,Y -474.718,Z 1076.550,A 0.000,B 0.000,C 90.000,E1 99.029} C_DIS
LIN {X -0.015,Y -474.652,Z 1076.547,A 0.000,B 0.000,C 90.000,E1 98.511} C_DIS
LIN {X 0.113,Y -473.601,Z 1076.544,A 0.000,B 0.000,C 90.000,E1 97.992} C_DIS
LIN {X -0.024,Y -472.661,Z 1076.543,A 0.000,B 0.000,C 90.000,E1 97.757} C_DIS
LIN {X -0.225,Y -471.387,Z 1076.542,A 0.000,B 0.000,C 90.000,E1 97.530} C_DIS
LIN {X 0.127,Y -460.743,Z 1076.533,A 0.000,B 0.000,C 90.000,E1 95.967} C_DIS
LIN {X -0.026,Y -451.759,Z 1076.526,A 0.000,B 0.000,C 90.000,E1 94.702} C_DIS
LIN {X 0.066,Y -439.527,Z 1076.516,A 0.000,B 0.000,C 90.000,E1 92.865} C_DIS
LIN {X -0.126,Y -423.466,Z 1076.501,A 0.000,B 0.000,C 90.000,E1 90.229} C_DIS
LIN {X 0.141,Y -406.936,Z 1076.484,A 0.000,B 0.000,C 90.000,E1 87.192} C_DIS
LIN {X 0.121,Y -397.958,Z 1076.475,A 0.000,B 0.000,C 90.000,E1 85.527} C_DIS
LIN {X -0.014,Y -387.214,Z 1076.464,A 0.000,B 0.000,C 90.000,E1 83.571} C_DIS
LIN {X 0.083,Y -377.917,Z 1076.455,A 0.000,B 0.000,C 90.000,E1 81.837} C_DIS
LIN {X 0.066,Y -368.343,Z 1076.445,A 0.000,B 0.000,C 90.000,E1 80.095} C_DIS
LIN {X -0.052,Y -358.454,Z 1076.435,A 0.000,B 0.000,C 90.000,E1 78.342} C_DIS
LIN {X 0.008,Y -346.825,Z 1076.423,A 0.000,B 0.000,C 90.000,E1 76.228} C_DIS
LIN {X -0.115,Y -333.636,Z 1076.410,A 0.000,B 0.000,C 90.000,E1 73.795} C_DIS
LIN {X 0.140,Y -317.857,Z 1076.392,A 0.000,B 0.000,C 90.000,E1 70.604} C_DIS
LIN {X 0.013,Y -306.048,Z 1076.378,A 0.000,B 0.000,C 90.000,E1 68.050} C_DIS
LIN {X 0.059,Y -294.643,Z 1076.363,A 0.000,B 0.000,C 90.000,E1 65.409} C_DIS
LIN {X -0.047,Y -283.421,Z 1076.349,A 0.000,B 0.000,C 90.000,E1 62.743} C_DIS
LIN {X -0.040,Y -272.500,Z 1076.333,A 0.000,B 0.000,C 90.000,E1 59.999} C_DIS
LIN {X 0.017,Y -260.574,Z 1076.316,A 0.000,B 0.000,C 90.000,E1 56.834} C_DIS
LIN {X -0.050,Y -249.171,Z 1076.298,A 0.000,B 0.000,C 90.000,E1 53.623} C_DIS
LIN {X 0.006,Y -238.347,Z 1076.280,A 0.000,B 0.000,C 90.000,E1 50.312} C_DIS
LIN {X 0.043,Y -229.324,Z 1076.263,A 0.000,B 0.000,C 90.000,E1 47.310} C_DIS
LIN {X 0.030,Y -220.867,Z 1076.246,A 0.000,B 0.000,C 90.000,E1 44.271} C_DIS
LIN {X 0.131,Y -212.791,Z 1076.229,A 0.000,B 0.000,C 90.000,E1 41.148} C_DIS
LIN {X 0.072,Y -205.120,Z 1076.211,A 0.000,B 0.000,C 90.000,E1 38.016} C_DIS
LIN {X 0.059,Y -198.056,Z 1076.193,A 0.000,B 0.000,C 90.000,E1 34.818} C_DIS
LIN {X -0.022,Y -191.638,Z 1076.175,A 0.000,B 0.000,C 90.000,E1 31.592} C_DIS
LIN {X 0.027,Y -185.948,Z 1076.157,A 0.000,B 0.000,C 90.000,E1 28.281} C_DIS
LIN {X 0.002,Y -181.008,Z 1076.139,A 0.000,B 0.000,C 90.000,E1 24.951} C_DIS
LIN {X -0.038,Y -176.749,Z 1076.120,A 0.000,B 0.000,C 90.000,E1 21.589} C_DIS
LIN {X -0.039,Y -173.150,Z 1076.101,A 0.000,B 0.000,C 90.000,E1 18.181} C_DIS
LIN {X -0.041,Y -169.679,Z 1076.077,A 0.000,B 0.000,C 90.000,E1 13.883} C_DIS
LIN {X -0.037,Y -166.863,Z 1076.048,A 0.000,B 0.000,C 90.000,E1 8.681} C_DIS
LIN {X 0.017,Y -167.606,Z 1075.949,A 0.000,B 0.000,C 90.000,E1 350.792} C_DIS
LIN {X -0.027,Y -170.316,Z 1075.925,A 0.000,B 0.000,C 90.000,E1 346.464} C_DIS
LIN {X 0.049,Y -174.091,Z 1075.901,A 0.000,B 0.000,C 90.000,E1 342.127} C_DIS
LIN {X 0.003,Y -177.870,Z 1075.882,A 0.000,B 0.000,C 90.000,E1 338.720} C_DIS
LIN {X -0.087,Y -182.327,Z 1075.863,A 0.000,B 0.000,C 90.000,E1 335.357} C_DIS
LIN {X -0.004,Y -187.479,Z 1075.844,A 0.000,B 0.000,C 90.000,E1 331.975} C_DIS
LIN {X -0.018,Y -193.533,Z 1075.826,A 0.000,B 0.000,C 90.000,E1 328.663} C_DIS
LIN {X -0.005,Y -200.393,Z 1075.808,A 0.000,B 0.000,C 90.000,E1 325.388} C_DIS
LIN {X -0.088,Y -207.938,Z 1075.790,A 0.000,B 0.000,C 90.000,E1 322.190} C_DIS
LIN {X 0.015,Y -217.277,Z 1075.770,A 0.000,B 0.000,C 90.000,E1 318.609} C_DIS
LIN {X 0.118,Y -226.338,Z 1075.753,A 0.000,B 0.000,C 90.000,E1 315.486} C_DIS
LIN {X 0.010,Y -235.122,Z 1075.738,A 0.000,B 0.000,C 90.000,E1 312.852} C_DIS
LIN {X -0.033,Y -243.545,Z 1075.726,A 0.000,B 0.000,C 90.000,E1 310.620} C_DIS
LIN {X 0.115,Y -252.973,Z 1075.713,A 0.000,B 0.000,C 90.000,E1 308.382} C_DIS
LIN {X -0.020,Y -263.510,Z 1075.701,A 0.000,B 0.000,C 90.000,E1 306.251} C_DIS
LIN {X 0.008,Y -280.781,Z 1075.684,A 0.000,B 0.000,C 90.000,E1 303.086} C_DIS
LIN {X 0.160,Y -299.508,Z 1075.667,A 0.000,B 0.000,C 90.000,E1 300.001} C_DIS
LIN {X 0.016,Y -319.732,Z 1075.650,A 0.000,B 0.000,C 90.000,E1 297.078} C_DIS
LIN {X -0.039,Y -334.105,Z 1075.640,A 0.000,B 0.000,C 90.000,E1 295.207} C_DIS
LIN {X -0.126,Y -347.197,Z 1075.631,A 0.000,B 0.000,C 90.000,E1 293.695} C_DIS
LIN {X 0.084,Y -366.235,Z 1075.621,A 0.000,B 0.000,C 90.000,E1 291.716} C_DIS
LIN {X -0.078,Y -391.135,Z 1075.608,A 0.000,B 0.000,C 90.000,E1 289.504} C_DIS
LIN {X 0.018,Y -404.958,Z 1075.602,A 0.000,B 0.000,C 90.000,E1 288.308} C_DIS
LIN {X 0.142,Y -415.690,Z 1075.596,A 0.000,B 0.000,C 90.000,E1 287.347} C_DIS
LIN {X 0.162,Y -423.529,Z 1075.592,A 0.000,B 0.000,C 90.000,E1 286.622} C_DIS
LIN {X -0.017,Y -431.119,Z 1075.588,A 0.000,B 0.000,C 90.000,E1 285.898} C_DIS
LIN {X 0.221,Y -440.940,Z 1075.583,A 0.000,B 0.000,C 90.000,E1 284.828} C_DIS
LIN {X 0.028,Y -447.904,Z 1075.578,A 0.000,B 0.000,C 90.000,E1 284.064} C_DIS
LIN {X -0.128,Y -454.338,Z 1075.574,A 0.000,B 0.000,C 90.000,E1 283.300} C_DIS
LIN {X -0.237,Y -460.120,Z 1075.569,A 0.000,B 0.000,C 90.000,E1 282.535} C_DIS
LIN {X 0.164,Y -465.181,Z 1075.565,A 0.000,B 0.000,C 90.000,E1 281.715} C_DIS
LIN {X 0.152,Y -469.426,Z 1075.561,A 0.000,B 0.000,C 90.000,E1 280.950} C_DIS
LIN {X 0.093,Y -473.075,Z 1075.557,A 0.000,B 0.000,C 90.000,E1 280.197} C_DIS
LIN {X 0.064,Y -476.122,Z 1075.552,A 0.000,B 0.000,C 90.000,E1 279.443} C_DIS
LIN {X -0.207,Y -477.843,Z 1075.550,A 0.000,B 0.000,C 90.000,E1 278.973} C_DIS
LIN {X -0.072,Y -479.343,Z 1075.547,A 0.000,B 0.000,C 90.000,E1 278.454} C_DIS
LIN {X 0.078,Y -480.614,Z 1075.544,A 0.000,B 0.000,C 90.000,E1 277.936} C_DIS
LIN {X -0.013,Y -482.628,Z 1075.539,A 0.000,B 0.000,C 90.000,E1 276.947} C_DIS
LIN {X 0.158,Y -483.307,Z 1075.536,A 0.000,B 0.000,C 90.000,E1 276.429} C_DIS
LIN {X -0.145,Y -483.724,Z 1075.533,A 0.000,B 0.000,C 90.000,E1 275.967} C_DIS
LIN {X -0.011,Y -483.810,Z 1075.530,A 0.000,B 0.000,C 90.000,E1 275.454} C_DIS
LIN {X 0.175,Y -483.404,Z 1075.528,A 0.000,B 0.000,C 90.000,E1 274.935} C_DIS
LIN {X -0.122,Y -482.626,Z 1075.525,A 0.000,B 0.000,C 90.000,E1 274.473} C_DIS
LIN {X 0.057,Y -481.294,Z 1075.522,A 0.000,B 0.000,C 90.000,E1 273.955} C_DIS
LIN {X 0.197,Y -479.383,Z 1075.519,A 0.000,B 0.000,C 90.000,E1 273.440} C_DIS
LIN {X -0.118,Y -476.778,Z 1075.516,A 0.000,B 0.000,C 90.000,E1 272.980} C_DIS
LIN {X 0.001,Y -473.447,Z 1075.514,A 0.000,B 0.000,C 90.000,E1 272.465} C_DIS
LIN {X 0.105,Y -469.152,Z 1075.511,A 0.000,B 0.000,C 90.000,E1 271.949} C_DIS
LIN {X -0.073,Y -466.650,Z 1075.510,A 0.000,B 0.000,C 90.000,E1 271.718} C_DIS
LIN {X 0.181,Y -461.057,Z 1075.507,A 0.000,B 0.000,C 90.000,E1 271.203} C_DIS
LIN {X -0.110,Y -454.989,Z 1075.504,A 0.000,B 0.000,C 90.000,E1 270.802} C_DIS
LIN {X 0.072,Y -451.709,Z 1075.503,A 0.000,B 0.000,C 90.000,E1 270.573} C_DIS
LIN {X -0.055,Y -444.691,Z 1075.501,A 0.000,B 0.000,C 90.000,E1 270.229} C_DIS
LIN {X -0.082,Y -437.203,Z 1075.500,A 0.000,B 0.000,C 90.000,E1 269.943} C_DIS
LIN {X -0.032,Y -429.527,Z 1075.498,A 0.000,B 0.000,C 90.000,E1 269.714} C_DIS
LIN {X -0.038,Y -421.461,Z 1075.497,A 0.000,B 0.000,C 90.000,E1 269.542} C_DIS
LIN {X -0.133,Y -412.367,Z 1075.497,A 0.000,B 0.000,C 90.000,E1 269.427} C_DIS
LIN {X 0.032,Y -402.508,Z 1075.496,A 0.000,B 0.000,C 90.000,E1 269.312} C_DIS
LIN {X 0.182,Y -392.965,Z 1075.496,A 0.000,B 0.000,C 90.000,E1 269.255} C_DIS
LIN {X 0.057,Y -181.383,Z 1075.496,A 0.000,B 0.000,C 90.000,E1 269.255} C_DIS
LIN {X 0.061,Y -180.907,Z 1075.475,A 0.000,B 0.000,C 90.000,E1 265.527} C_DIS
LIN {X -0.062,Y -180.769,Z 1075.471,A 0.000,B 0.000,C 90.000,E1 264.723} C_DIS
LIN {X 0.010,Y -178.864,Z 1075.442,A 0.000,B 0.000,C 90.000,E1 259.634} C_DIS
LIN {X -0.089,Y -175.907,Z 1075.414,A 0.000,B 0.000,C 90.000,E1 254.574} C_DIS
LIN {X 0.019,Y -174.591,Z 1075.405,A 0.000,B 0.000,C 90.000,E1 252.834} C_DIS
LIN {X 0.054,Y -171.573,Z 1075.381,A 0.000,B 0.000,C 90.000,E1 248.539} C_DIS
LIN {X 0.035,Y -167.796,Z 1075.357,A 0.000,B 0.000,C 90.000,E1 244.229} C_DIS
LIN {X 0.050,Y -166.514,Z 1075.347,A 0.000,B 0.000,C 90.000,E1 242.487} C_DIS
LIN {X 0.045,Y -163.222,Z 1075.328,A 0.000,B 0.000,C 90.000,E1 238.997} C_DIS
LIN {X 0.009,Y -161.187,Z 1075.313,A 0.000,B 0.000,C 90.000,E1 236.373} C_DIS
LIN {X 0.009,Y -157.199,Z 1075.289,A 0.000,B 0.000,C 90.000,E1 231.949} C_DIS
LIN {X 0.055,Y -155.928,Z 1075.279,A 0.000,B 0.000,C 90.000,E1 230.150} C_DIS
LIN {X 0.005,Y -152.179,Z 1075.254,A 0.000,B 0.000,C 90.000,E1 225.688} C_DIS
LIN {X 0.020,Y -150.426,Z 1075.239,A 0.000,B 0.000,C 90.000,E1 222.975} C_DIS
LIN {X -0.055,Y -147.154,Z 1075.214,A 0.000,B 0.000,C 90.000,E1 218.463} C_DIS
LIN {X 0.032,Y -145.168,Z 1075.193,A 0.000,B 0.000,C 90.000,E1 214.771} C_DIS
LIN {X -0.051,Y -142.320,Z 1075.163,A 0.000,B 0.000,C 90.000,E1 209.283} C_DIS
LIN {X 0.069,Y -141.709,Z 1075.152,A 0.000,B 0.000,C 90.000,E1 207.385} C_DIS
LIN {X -0.008,Y -139.470,Z 1075.116,A 0.000,B 0.000,C 90.000,E1 200.918} C_DIS
LIN {X 0.045,Y -139.203,Z 1075.106,A 0.000,B 0.000,C 90.000,E1 199.033} C_DIS
LIN {X -0.028,Y -138.328,Z 1075.054,A 0.000,B 0.000,C 90.000,E1 189.726} C_DIS
LIN {X -0.025,Y -139.440,Z 1075.007,A 0.000,B 0.000,C 90.000,E1 181.318} C_DIS
LIN {X 0.055,Y -140.974,Z 1074.976,A 0.000,B 0.000,C 90.000,E1 175.698} C_DIS
LIN {X 0.005,Y -142.730,Z 1074.956,A 0.000,B 0.000,C 90.000,E1 172.008} C_DIS
LIN {X -0.037,Y -145.116,Z 1074.930,A 0.000,B 0.000,C 90.000,E1 167.409} C_DIS
LIN {X -0.044,Y -147.740,Z 1074.910,A 0.000,B 0.000,C 90.000,E1 163.740} C_DIS
LIN {X 0.038,Y -150.405,Z 1074.889,A 0.000,B 0.000,C 90.000,E1 160.061} C_DIS
LIN {X -0.087,Y -153.842,Z 1074.869,A 0.000,B 0.000,C 90.000,E1 156.485} C_DIS
LIN {X -0.028,Y -157.253,Z 1074.849,A 0.000,B 0.000,C 90.000,E1 152.871} C_DIS
LIN {X 0.050,Y -161.426,Z 1074.829,A 0.000,B 0.000,C 90.000,E1 149.282} C_DIS
LIN {X -0.079,Y -165.628,Z 1074.810,A 0.000,B 0.000,C 90.000,E1 145.801} C_DIS
LIN {X 0.040,Y -170.557,Z 1074.791,A 0.000,B 0.000,C 90.000,E1 142.271} C_DIS
LIN {X -0.052,Y -175.436,Z 1074.771,A 0.000,B 0.000,C 90.000,E1 138.852} C_DIS
LIN {X 0.064,Y -181.060,Z 1074.752,A 0.000,B 0.000,C 90.000,E1 135.405} C_DIS
LIN {X -0.070,Y -186.496,Z 1074.734,A 0.000,B 0.000,C 90.000,E1 132.081} C_DIS
LIN {X -0.002,Y -191.117,Z 1074.720,A 0.000,B 0.000,C 90.000,E1 129.564} C_DIS
LIN {X -0.082,Y -196.911,Z 1074.702,A 0.000,B 0.000,C 90.000,E1 126.297} C_DIS
LIN {X 0.007,Y -199.125,Z 1074.695,A 0.000,B 0.000,C 90.000,E1 125.152} C_DIS
LIN {X -0.037,Y -306.517,Z 1074.695,A 0.000,B 0.000,C 90.000,E1 125.152} C_DIS
LIN {X -0.044,Y -312.632,Z 1074.694,A 0.000,B 0.000,C 90.000,E1 124.898} C_DIS
LIN {X 0.179,Y -315.408,Z 1074.693,A 0.000,B 0.000,C 90.000,E1 124.612} C_DIS
LIN {X 0.087,Y -319.159,Z 1074.690,A 0.000,B 0.000,C 90.000,E1 124.119} C_DIS
LIN {X 0.153,Y -320.817,Z 1074.688,A 0.000,B 0.000,C 90.000,E1 123.785} C_DIS
LIN {X 0.036,Y -323.210,Z 1074.684,A 0.000,B 0.000,C 90.000,E1 123.166} C_DIS
LIN {X -0.043,Y -333.661,Z 1074.668,A 0.000,B 0.000,C 90.000,E1 120.335} C_DIS
LIN {X 0.136,Y -345.459,Z 1074.653,A 0.000,B 0.000,C 90.000,E1 117.513} C_DIS
LIN {X 0.178,Y -358.714,Z 1074.638,A 0.000,B 0.000,C 90.000,E1 114.771} C_DIS
LIN {X 0.068,Y -371.808,Z 1074.625,A 0.000,B 0.000,C 90.000,E1 112.408} C_DIS
LIN {X 0.150,Y -386.234,Z 1074.612,A 0.000,B 0.000,C 90.000,E1 110.066} C_DIS
LIN {X -0.049,Y -402.094,Z 1074.599,A 0.000,B 0.000,C 90.000,E1 107.819} C_DIS
LIN {X -0.115,Y -419.501,Z 1074.587,A 0.000,B 0.000,C 90.000,E1 105.607} C_DIS
LIN {X 0.142,Y -438.573,Z 1074.575,A 0.000,B 0.000,C 90.000,E1 103.411} C_DIS
LIN {X -0.144,Y -458.657,Z 1074.563,A 0.000,B 0.000,C 90.000,E1 101.422} C_DIS
LIN {X 0.179,Y -468.716,Z 1074.558,A 0.000,B 0.000,C 90.000,E1 100.433} C_DIS
LIN {X 0.106,Y -470.600,Z 1074.557,A 0.000,B 0.000,C 90.000,E1 100.197} C_DIS
LIN {X 0.032,Y -472.027,Z 1074.555,A 0.000,B 0.000,C 90.000,E1 99.962} C_DIS
LIN {X 0.133,Y -473.932,Z 1074.553,A 0.000,B 0.000,C 90.000,E1 99.443} C_DIS
LIN {X -0.149,Y -474.727,Z 1074.550,A 0.000,B 0.000,C 90.000,E1 98.973} C_DIS
LIN {X -0.027,Y -474.551,Z 1074.547,A 0.000,B 0.000,C 90.000,E1 98.454} C_DIS
LIN {X 0.103,Y -473.379,Z 1074.544,A 0.000,B 0.000,C 90.000,E1 97.936} C_DIS
LIN {X -0.035,Y -472.366,Z 1074.543,A 0.000,B 0.000,C 90.000,E1 97.701} C_DIS
LIN {X -0.175,Y -471.004,Z 1074.541,A 0.000,B 0.000,C 90.000,E1 97.466} C_DIS
LIN {X 0.162,Y -456.779,Z 1074.530,A 0.000,B 0.000,C 90.000,E1 95.391} C_DIS
LIN {X 0.092,Y -442.495,Z 1074.519,A 0.000,B 0.000,C 90.000,E1 93.326} C_DIS
LIN {X 0.129,Y -424.663,Z 1074.502,A 0.000,B 0.000,C 90.000,E1 90.401} C_DIS
LIN {X 0.092,Y -406.605,Z 1074.484,A 0.000,B 0.000,C 90.000,E1 87.135} C_DIS
LIN {X 0.067,Y -397.619,Z 1074.475,A 0.000,B 0.000,C 90.000,E1 85.469} C_DIS
LIN {X -0.074,Y -386.857,Z 1074.464,A 0.000,B 0.000,C 90.000,E1 83.514} C_DIS
LIN {X 0.016,Y -377.526,Z 1074.454,A 0.000,B 0.000,C 90.000,E1 81.781} C_DIS
LIN {X -0.008,Y -367.943,Z 1074.445,A 0.000,B 0.000,C 90.000,E1 80.038} C_DIS
LIN {X -0.133,Y -358.017,Z 1074.435,A 0.000,B 0.000,C 90.000,E1 78.285} C_DIS
LIN {X -0.082,Y -346.387,Z 1074.423,A 0.000,B 0.000,C 90.000,E1 76.172} C_DIS
LIN {X 0.104,Y -333.227,Z 1074.409,A 0.000,B 0.000,C 90.000,E1 73.685} C_DIS
LIN {X 0.088,Y -319.026,Z 1074.394,A 0.000,B 0.000,C 90.000,E1 70.859} C_DIS
LIN {X 0.097,Y -307.141,Z 1074.379,A 0.000,B 0.000,C 90.000,E1 68.284} C_DIS
LIN {X 0.051,Y -295.698,Z 1074.365,A 0.000,B 0.000,C 90.000,E1 65.665} C_DIS
LIN {X -0.028,Y -284.447,Z 1074.350,A 0.000,B 0.000,C 90.000,E1 62.999} C_DIS
LIN {X 0.005,Y -273.487,Z 1074.335,A 0.000,B 0.000,C 90.000,E1 60.255} C_DIS
LIN {X -0.055,Y -261.504,Z 1074.317,A 0.000,B 0.000,C 90.000,E1 57.120} C_DIS
LIN {X -0.093,Y -250.022,Z 1074.299,A 0.000,B 0.000,C 90.000,E1 53.909} C_DIS
LIN {X -0.013,Y -239.109,Z 1074.281,A 0.000,B 0.000,C 90.000,E1 50.598} C_DIS
LIN {X 0.003,Y -228.898,Z 1074.262,A 0.000,B 0.000,C 90.000,E1 47.229} C_DIS
LIN {X -0.020,Y -220.430,Z 1074.245,A 0.000,B 0.000,C 90.000,E1 44.190} C_DIS
LIN {X 0.073,Y -212.356,Z 1074.228,A 0.000,B 0.000,C 90.000,E1 41.067} C_DIS
LIN {X 0.002,Y -204.699,Z 1074.211,A 0.000,B 0.000,C 90.000,E1 37.935} C_DIS
LIN {X -0.020,Y -197.632,Z 1074.193,A 0.000,B 0.000,C 90.000,E1 34.739} C_DIS
LIN {X 0.051,Y -191.255,Z 1074.175,A 0.000,B 0.000,C 90.000,E1 31.465} C_DIS
LIN {X 0.003,Y -185.600,Z 1074.157,A 0.000,B 0.000,C 90.000,E1 28.180} C_DIS
LIN {X -0.021,Y -180.654,Z 1074.138,A 0.000,B 0.000,C 90.000,E1 24.847} C_DIS
LIN {X 0.005,Y -176.422,Z 1074.119,A 0.000,B 0.000,C 90.000,E1 21.461} C_DIS
LIN {X -0.008,Y -172.851,Z 1074.100,A 0.000,B 0.000,C 90.000,E1 18.055} C_DIS
LIN {X -0.064,Y -169.404,Z 1074.076,A 0.000,B 0.000,C 90.000,E1 13.772} C_DIS
LIN {X -0.063,Y -166.616,Z 1074.047,A 0.000,B 0.000,C 90.000,E1 8.568} C_DIS
LIN {X 0.005,Y -167.414,Z 1073.949,A 0.000,B 0.000,C 90.000,E1 350.792} C_DIS
LIN {X -0.045,Y -170.142,Z 1073.925,A 0.000,B 0.000,C 90.000,E1 346.464} C_DIS
LIN {X 0.025,Y -173.901,Z 1073.901,A 0.000,B 0.000,C 90.000,E1 342.127} C_DIS
LIN {X -0.025,Y -177.692,Z 1073.882,A 0.000,B 0.000,C 90.000,E1 338.720} C_DIS
LIN {X 0.045,Y -182.170,Z 1073.863,A 0.000,B 0.000,C 90.000,E1 335.305} C_DIS
LIN {X -0.043,Y -187.326,Z 1073.844,A 0.000,B 0.000,C 90.000,E1 331.975} C_DIS
LIN {X -0.062,Y -193.393,Z 1073.826,A 0.000,B 0.000,C 90.000,E1 328.663} C_DIS
LIN {X -0.053,Y -200.267,Z 1073.808,A 0.000,B 0.000,C 90.000,E1 325.388} C_DIS
LIN {X 0.022,Y -207.817,Z 1073.790,A 0.000,B 0.000,C 90.000,E1 322.145} C_DIS
LIN {X -0.045,Y -217.183,Z 1073.770,A 0.000,B 0.000,C 90.000,E1 318.609} C_DIS
LIN {X 0.054,Y -226.242,Z 1073.753,A 0.000,B 0.000,C 90.000,E1 315.486} C_DIS
LIN {X -0.058,Y -234.990,Z 1073.738,A 0.000,B 0.000,C 90.000,E1 312.852} C_DIS
LIN {X 0.039,Y -244.899,Z 1073.724,A 0.000,B 0.000,C 90.000,E1 310.216} C_DIS
LIN {X 0.036,Y -252.821,Z 1073.713,A 0.000,B 0.000,C 90.000,E1 308.382} C_DIS
LIN {X 0.051,Y -263.405,Z 1073.701,A 0.000,B 0.000,C 90.000,E1 306.217} C_DIS
LIN {X -0.086,Y -280.721,Z 1073.684,A 0.000,B 0.000,C 90.000,E1 303.086} C_DIS
LIN {X 0.059,Y -299.459,Z 1073.667,A 0.000,B 0.000,C 90.000,E1 300.001} C_DIS
LIN {X 0.053,Y -319.727,Z 1073.650,A 0.000,B 0.000,C 90.000,E1 297.052} C_DIS
LIN {X 0.017,Y -331.820,Z 1073.641,A 0.000,B 0.000,C 90.000,E1 295.463} C_DIS
LIN {X -0.152,Y -344.845,Z 1073.633,A 0.000,B 0.000,C 90.000,E1 293.951} C_DIS
LIN {X -0.036,Y -363.807,Z 1073.622,A 0.000,B 0.000,C 90.000,E1 291.972} C_DIS
LIN {X -0.061,Y -391.139,Z 1073.608,A 0.000,B 0.000,C 90.000,E1 289.504} C_DIS
LIN {X 0.154,Y -404.773,Z 1073.602,A 0.000,B 0.000,C 90.000,E1 288.308} C_DIS
LIN {X -0.110,Y -415.520,Z 1073.597,A 0.000,B 0.000,C 90.000,E1 287.402} C_DIS
LIN {X -0.107,Y -423.347,Z 1073.593,A 0.000,B 0.000,C 90.000,E1 286.677} C_DIS
LIN {X 0.116,Y -430.947,Z 1073.588,A 0.000,B 0.000,C 90.000,E1 285.898} C_DIS
LIN {X -0.168,Y -440.776,Z 1073.583,A 0.000,B 0.000,C 90.000,E1 284.898} C_DIS
LIN {X 0.192,Y -447.744,Z 1073.578,A 0.000,B 0.000,C 90.000,E1 284.064} C_DIS
LIN {X 0.036,Y -454.183,Z 1073.574,A 0.000,B 0.000,C 90.000,E1 283.300} C_DIS
LIN {X -0.072,Y -459.988,Z 1073.570,A 0.000,B 0.000,C 90.000,E1 282.535} C_DIS
LIN {X 0.037,Y -463.498,Z 1073.567,A 0.000,B 0.000,C 90.000,E1 282.007} C_DIS
LIN {X 0.014,Y -468.024,Z 1073.563,A 0.000,B 0.000,C 90.000,E1 281.243} C_DIS
LIN {X -0.064,Y -471.887,Z 1073.558,A 0.000,B 0.000,C 90.000,E1 280.489} C_DIS
LIN {X 0.119,Y -474.159,Z 1073.555,A 0.000,B 0.000,C 90.000,E1 279.962} C_DIS
LIN {X -0.237,Y -476.155,Z 1073.553,A 0.000,B 0.000,C 90.000,E1 279.500} C_DIS
LIN {X -0.038,Y -477.911,Z 1073.550,A 0.000,B 0.000,C 90.000,E1 278.973} C_DIS
LIN {X 0.098,Y -479.429,Z 1073.547,A 0.000,B 0.000,C 90.000,E1 278.454} C_DIS
LIN {X -0.005,Y -481.858,Z 1073.542,A 0.000,B 0.000,C 90.000,E1 277.466} C_DIS
LIN {X 0.160,Y -482.815,Z 1073.539,A 0.000,B 0.000,C 90.000,E1 276.947} C_DIS
LIN {X -0.148,Y -483.547,Z 1073.536,A 0.000,B 0.000,C 90.000,E1 276.486} C_DIS
LIN {X 0.030,Y -483.993,Z 1073.533,A 0.000,B 0.000,C 90.000,E1 275.967} C_DIS
LIN {X 0.166,Y -484.074,Z 1073.530,A 0.000,B 0.000,C 90.000,E1 275.454} C_DIS
LIN {X -0.129,Y -483.742,Z 1073.528,A 0.000,B 0.000,C 90.000,E1 274.992} C_DIS
LIN {X 0.056,Y -482.981,Z 1073.525,A 0.000,B 0.000,C 90.000,E1 274.473} C_DIS
LIN {X 0.237,Y -481.682,Z 1073.522,A 0.000,B 0.000,C 90.000,E1 273.955} C_DIS
LIN {X -0.099,Y -479.758,Z 1073.519,A 0.000,B 0.000,C 90.000,E1 273.498} C_DIS
LIN {X 0.065,Y -477.200,Z 1073.517,A 0.000,B 0.000,C 90.000,E1 272.980} C_DIS
LIN {X 0.186,Y -473.927,Z 1073.514,A 0.000,B 0.000,C 90.000,E1 272.465} C_DIS
LIN {X -0.180,Y -469.717,Z 1073.511,A 0.000,B 0.000,C 90.000,E1 272.007} C_DIS
LIN {X -0.079,Y -464.423,Z 1073.508,A 0.000,B 0.000,C 90.000,E1 271.489} C_DIS
LIN {X -0.148,Y -458.623,Z 1073.506,A 0.000,B 0.000,C 90.000,E1 271.031} C_DIS
LIN {X 0.180,Y -452.320,Z 1073.503,A 0.000,B 0.000,C 90.000,E1 270.573} C_DIS
LIN {X 0.117,Y -449.138,Z 1073.502,A 0.000,B 0.000,C 90.000,E1 270.401} C_DIS
LIN {X -0.182,Y -442.099,Z 1073.500,A 0.000,B 0.000,C 90.000,E1 270.115} C_DIS
LIN {X 0.003,Y -434.642,Z 1073.499,A 0.000,B 0.000,C 90.000,E1 269.828} C_DIS
LIN {X 0.187,Y -426.645,Z 1073.498,A 0.000,B 0.000,C 90.000,E1 269.599} C_DIS
LIN {X -0.090,Y -418.604,Z 1073.497,A 0.000,B 0.000,C 90.000,E1 269.484} C_DIS
LIN {X -0.055,Y -409.460,Z 1073.496,A 0.000,B 0.000,C 90.000,E1 269.370} C_DIS
LIN {X -0.097,Y -401.864,Z 1073.496,A 0.000,B 0.000,C 90.000,E1 269.312} C_DIS
LIN {X 0.111,Y -394.510,Z 1073.496,A 0.000,B 0.000,C 90.000,E1 269.255} C_DIS
LIN {X 0.023,Y -181.380,Z 1073.496,A 0.000,B 0.000,C 90.000,E1 269.255} C_DIS
LIN {X 0.053,Y -180.908,Z 1073.475,A 0.000,B 0.000,C 90.000,E1 265.527} C_DIS
LIN {X -0.070,Y -180.768,Z 1073.471,A 0.000,B 0.000,C 90.000,E1 264.723} C_DIS
LIN {X 0.002,Y -178.862,Z 1073.442,A 0.000,B 0.000,C 90.000,E1 259.634} C_DIS
LIN {X 0.072,Y -175.905,Z 1073.414,A 0.000,B 0.000,C 90.000,E1 254.519} C_DIS
LIN {X 0.010,Y -174.588,Z 1073.405,A 0.000,B 0.000,C 90.000,E1 252.834} C_DIS
LIN {X 0.046,Y -171.571,Z 1073.381,A 0.000,B 0.000,C 90.000,E1 248.539} C_DIS
LIN {X 0.028,Y -167.794,Z 1073.357,A 0.000,B 0.000,C 90.000,E1 244.229} C_DIS
LIN {X 0.043,Y -166.511,Z 1073.347,A 0.000,B 0.000,C 90.000,E1 242.487} C_DIS
LIN {X 0.038,Y -163.219,Z 1073.328,A 0.000,B 0.000,C 90.000,E1 238.997} C_DIS
LIN {X 0.002,Y -161.185,Z 1073.313,A 0.000,B 0.000,C 90.000,E1 236.373} C_DIS
LIN {X 0.002,Y -157.197,Z 1073.289,A 0.000,B 0.000,C 90.000,E1 231.949} C_DIS
LIN {X 0.048,Y -155.925,Z 1073.279,A 0.000,B 0.000,C 90.000,E1 230.150} C_DIS
LIN {X -0.003,Y -152.177,Z 1073.254,A 0.000,B 0.000,C 90.000,E1 225.688} C_DIS
LIN {X 0.012,Y -150.424,Z 1073.239,A 0.000,B 0.000,C 90.000,E1 222.975} C_DIS
LIN {X -0.061,Y -147.152,Z 1073.214,A 0.000,B 0.000,C 90.000,E1 218.463} C_DIS
LIN {X 0.025,Y -145.167,Z 1073.193,A 0.000,B 0.000,C 90.000,E1 214.771} C_DIS
LIN {X -0.058,Y -142.318,Z 1073.163,A 0.000,B 0.000,C 90.000,E1 209.283} C_DIS
LIN {X 0.062,Y -141.708,Z 1073.152,A 0.000,B 0.000,C 90.000,E1 207.385} C_DIS
LIN {X -0.015,Y -139.470,Z 1073.116,A 0.000,B 0.000,C 90.000,E1 200.918} C_DIS
LIN {X 0.038,Y -139.203,Z 1073.106,A 0.000,B 0.000,C 90.000,E1 199.033} C_DIS
LIN {X -0.035,Y -138.328,Z 1073.054,A 0.000,B 0.000,C 90.000,E1 189.726} C_DIS
LIN {X -0.032,Y -139.441,Z 1073.007,A 0.000,B 0.000,C 90.000,E1 181.318} C_DIS
LIN {X 0.048,Y -140.976,Z 1072.976,A 0.000,B 0.000,C 90.000,E1 175.698} C_DIS
LIN {X -0.002,Y -142.731,Z 1072.956,A 0.000,B 0.000,C 90.000,E1 172.008} C_DIS
LIN {X -0.045,Y -145.118,Z 1072.930,A 0.000,B 0.000,C 90.000,E1 167.409} C_DIS
LIN {X -0.050,Y -147.742,Z 1072.910,A 0.000,B 0.000,C 90.000,E1 163.740} C_DIS
LIN {X 0.031,Y -150.408,Z 1072.889,A 0.000,B 0.000,C 90.000,E1 160.061} C_DIS
LIN {X 0.047,Y -153.845,Z 1072.869,A 0.000,B 0.000,C 90.000,E1 156.433} C_DIS
LIN {X -0.036,Y -157.256,Z 1072.849,A 0.000,B 0.000,C 90.000,E1 152.871} C_DIS
LIN {X 0.042,Y -161.430,Z 1072.829,A 0.000,B 0.000,C 90.000,E1 149.282} C_DIS
LIN {X 0.049,Y -165.631,Z 1072.810,A 0.000,B 0.000,C 90.000,E1 145.754} C_DIS
LIN {X 0.032,Y -170.562,Z 1072.790,A 0.000,B 0.000,C 90.000,E1 142.271} C_DIS
LIN {X -0.060,Y -175.439,Z 1072.771,A 0.000,B 0.000,C 90.000,E1 138.852} C_DIS
LIN {X 0.057,Y -181.063,Z 1072.752,A 0.000,B 0.000,C 90.000,E1 135.405} C_DIS
LIN {X -0.078,Y -186.501,Z 1072.734,A 0.000,B 0.000,C 90.000,E1 132.081} C_DIS
LIN {X -0.010,Y -191.120,Z 1072.720,A 0.000,B 0.000,C 90.000,E1 129.564} C_DIS
LIN {X -0.090,Y -196.916,Z 1072.702,A 0.000,B 0.000,C 90.000,E1 126.297} C_DIS
LIN {X 0.069,Y -199.021,Z 1072.696,A 0.000,B 0.000,C 90.000,E1 125.185} C_DIS
LIN {X 0.058,Y -305.773,Z 1072.696,A 0.000,B 0.000,C 90.000,E1 125.185} C_DIS
LIN {X 0.175,Y -310.509,Z 1072.695,A 0.000,B 0.000,C 90.000,E1 125.025} C_DIS
LIN {X 0.112,Y -312.701,Z 1072.694,A 0.000,B 0.000,C 90.000,E1 124.898} C_DIS
LIN {X 0.166,Y -315.687,Z 1072.693,A 0.000,B 0.000,C 90.000,E1 124.612} C_DIS
LIN {X -0.034,Y -319.370,Z 1072.690,A 0.000,B 0.000,C 90.000,E1 124.119} C_DIS
LIN {X 0.033,Y -320.942,Z 1072.688,A 0.000,B 0.000,C 90.000,E1 123.785} C_DIS
LIN {X -0.179,Y -325.474,Z 1072.681,A 0.000,B 0.000,C 90.000,E1 122.546} C_DIS
LIN {X 0.086,Y -336.226,Z 1072.665,A 0.000,B 0.000,C 90.000,E1 119.667} C_DIS
LIN {X 0.179,Y -348.349,Z 1072.649,A 0.000,B 0.000,C 90.000,E1 116.873} C_DIS
LIN {X -0.172,Y -361.952,Z 1072.634,A 0.000,B 0.000,C 90.000,E1 114.207} C_DIS
LIN {X -0.213,Y -375.381,Z 1072.621,A 0.000,B 0.000,C 90.000,E1 111.844} C_DIS
LIN {X -0.060,Y -390.168,Z 1072.608,A 0.000,B 0.000,C 90.000,E1 109.504} C_DIS
LIN {X 0.082,Y -406.416,Z 1072.596,A 0.000,B 0.000,C 90.000,E1 107.221} C_DIS
LIN {X 0.128,Y -424.243,Z 1072.583,A 0.000,B 0.000,C 90.000,E1 105.009} C_DIS
LIN {X 0.046,Y -443.683,Z 1072.572,A 0.000,B 0.000,C 90.000,E1 102.883} C_DIS
LIN {X 0.112,Y -463.913,Z 1072.561,A 0.000,B 0.000,C 90.000,E1 100.894} C_DIS
LIN {X 0.047,Y -468.827,Z 1072.558,A 0.000,B 0.000,C 90.000,E1 100.433} C_DIS
LIN {X -0.044,Y -470.690,Z 1072.557,A 0.000,B 0.000,C 90.000,E1 100.197} C_DIS
LIN {X -0.137,Y -472.099,Z 1072.555,A 0.000,B 0.000,C 90.000,E1 99.962} C_DIS
LIN {X -0.037,Y -473.953,Z 1072.552,A 0.000,B 0.000,C 90.000,E1 99.443} C_DIS
LIN {X 0.149,Y -474.707,Z 1072.550,A 0.000,B 0.000,C 90.000,E1 98.916} C_DIS
LIN {X -0.197,Y -474.491,Z 1072.547,A 0.000,B 0.000,C 90.000,E1 98.454} C_DIS
LIN {X -0.067,Y -473.276,Z 1072.544,A 0.000,B 0.000,C 90.000,E1 97.936} C_DIS
LIN {X -0.204,Y -472.237,Z 1072.543,A 0.000,B 0.000,C 90.000,E1 97.701} C_DIS
LIN {X 0.124,Y -470.844,Z 1072.541,A 0.000,B 0.000,C 90.000,E1 97.409} C_DIS
LIN {X -0.005,Y -456.595,Z 1072.530,A 0.000,B 0.000,C 90.000,E1 95.391} C_DIS
LIN {X -0.073,Y -442.345,Z 1072.518,A 0.000,B 0.000,C 90.000,E1 93.326} C_DIS
LIN {X -0.035,Y -424.520,Z 1072.502,A 0.000,B 0.000,C 90.000,E1 90.401} C_DIS
LIN {X -0.069,Y -406.481,Z 1072.484,A 0.000,B 0.000,C 90.000,E1 87.135} C_DIS
LIN {X -0.093,Y -397.499,Z 1072.475,A 0.000,B 0.000,C 90.000,E1 85.469} C_DIS
LIN {X 0.152,Y -386.751,Z 1072.464,A 0.000,B 0.000,C 90.000,E1 83.457} C_DIS
LIN {X -0.141,Y -377.386,Z 1072.454,A 0.000,B 0.000,C 90.000,E1 81.781} C_DIS
LIN {X -0.163,Y -367.778,Z 1072.444,A 0.000,B 0.000,C 90.000,E1 80.038} C_DIS
LIN {X 0.064,Y -357.846,Z 1072.435,A 0.000,B 0.000,C 90.000,E1 78.229} C_DIS
LIN {X 0.102,Y -346.196,Z 1072.423,A 0.000,B 0.000,C 90.000,E1 76.117} C_DIS
LIN {X -0.047,Y -333.083,Z 1072.409,A 0.000,B 0.000,C 90.000,E1 73.685} C_DIS
LIN {X -0.120,Y -317.377,Z 1072.392,A 0.000,B 0.000,C 90.000,E1 70.550} C_DIS
LIN {X -0.140,Y -305.535,Z 1072.377,A 0.000,B 0.000,C 90.000,E1 67.975} C_DIS
LIN {X 0.050,Y -294.129,Z 1072.363,A 0.000,B 0.000,C 90.000,E1 65.305} C_DIS
LIN {X 0.052,Y -282.894,Z 1072.348,A 0.000,B 0.000,C 90.000,E1 62.615} C_DIS
LIN {X 0.041,Y -271.976,Z 1072.333,A 0.000,B 0.000,C 90.000,E1 59.871} C_DIS
LIN {X 0.075,Y -260.020,Z 1072.315,A 0.000,B 0.000,C 90.000,E1 56.707} C_DIS
LIN {X -0.013,Y -248.574,Z 1072.297,A 0.000,B 0.000,C 90.000,E1 53.497} C_DIS
LIN {X -0.013,Y -237.710,Z 1072.279,A 0.000,B 0.000,C 90.000,E1 50.194} C_DIS
LIN {X 0.033,Y -228.637,Z 1072.262,A 0.000,B 0.000,C 90.000,E1 47.187} C_DIS
LIN {X -0.005,Y -220.149,Z 1072.245,A 0.000,B 0.000,C 90.000,E1 44.150} C_DIS
LIN {X -0.068,Y -212.075,Z 1072.228,A 0.000,B 0.000,C 90.000,E1 41.067} C_DIS
LIN {X 0.021,Y -204.423,Z 1072.211,A 0.000,B 0.000,C 90.000,E1 37.890} C_DIS
LIN {X -0.002,Y -197.354,Z 1072.193,A 0.000,B 0.000,C 90.000,E1 34.692} C_DIS
LIN {X -0.095,Y -190.990,Z 1072.175,A 0.000,B 0.000,C 90.000,E1 31.465} C_DIS
LIN {X -0.058,Y -185.350,Z 1072.156,A 0.000,B 0.000,C 90.000,E1 28.153} C_DIS
LIN {X 0.068,Y -180.389,Z 1072.138,A 0.000,B 0.000,C 90.000,E1 24.771} C_DIS
LIN {X 0.015,Y -176.170,Z 1072.119,A 0.000,B 0.000,C 90.000,E1 21.408} C_DIS
LIN {X 0.001,Y -172.615,Z 1072.100,A 0.000,B 0.000,C 90.000,E1 18.000} C_DIS
LIN {X -0.019,Y -169.177,Z 1072.076,A 0.000,B 0.000,C 90.000,E1 13.703} C_DIS
LIN {X -0.064,Y -166.400,Z 1072.047,A 0.000,B 0.000,C 90.000,E1 8.511} C_DIS
LIN {X -0.006,Y -167.226,Z 1071.949,A 0.000,B 0.000,C 90.000,E1 350.792} C_DIS
LIN {X -0.061,Y -169.969,Z 1071.925,A 0.000,B 0.000,C 90.000,E1 346.464} C_DIS
LIN {X 0.003,Y -173.737,Z 1071.901,A 0.000,B 0.000,C 90.000,E1 342.127} C_DIS
LIN {X -0.053,Y -177.519,Z 1071.882,A 0.000,B 0.000,C 90.000,E1 338.720} C_DIS
LIN {X 0.013,Y -182.012,Z 1071.863,A 0.000,B 0.000,C 90.000,E1 335.305} C_DIS
LIN {X -0.079,Y -187.174,Z 1071.844,A 0.000,B 0.000,C 90.000,E1 331.975} C_DIS
LIN {X 0.062,Y -193.258,Z 1071.826,A 0.000,B 0.000,C 90.000,E1 328.614} C_DIS
LIN {X -0.100,Y -200.152,Z 1071.807,A 0.000,B 0.000,C 90.000,E1 325.388} C_DIS
LIN {X 0.099,Y -207.711,Z 1071.790,A 0.000,B 0.000,C 90.000,E1 322.110} C_DIS
LIN {X 0.068,Y -217.078,Z 1071.770,A 0.000,B 0.000,C 90.000,E1 318.566} C_DIS
LIN {X -0.001,Y -226.139,Z 1071.753,A 0.000,B 0.000,C 90.000,E1 315.486} C_DIS
LIN {X -0.118,Y -234.860,Z 1071.738,A 0.000,B 0.000,C 90.000,E1 312.852} C_DIS
LIN {X -0.026,Y -244.757,Z 1071.723,A 0.000,B 0.000,C 90.000,E1 310.216} C_DIS
LIN {X -0.033,Y -252.677,Z 1071.713,A 0.000,B 0.000,C 90.000,E1 308.382} C_DIS
LIN {X -0.130,Y -265.157,Z 1071.699,A 0.000,B 0.000,C 90.000,E1 305.884} C_DIS
LIN {X 0.010,Y -282.657,Z 1071.682,A 0.000,B 0.000,C 90.000,E1 302.704} C_DIS
LIN {X -0.024,Y -301.570,Z 1071.665,A 0.000,B 0.000,C 90.000,E1 299.667} C_DIS
LIN {X -0.129,Y -322.034,Z 1071.648,A 0.000,B 0.000,C 90.000,E1 296.744} C_DIS
LIN {X -0.020,Y -336.797,Z 1071.638,A 0.000,B 0.000,C 90.000,E1 294.847} C_DIS
LIN {X -0.098,Y -347.520,Z 1071.631,A 0.000,B 0.000,C 90.000,E1 293.643} C_DIS
LIN {X 0.008,Y -366.408,Z 1071.621,A 0.000,B 0.000,C 90.000,E1 291.716} C_DIS
LIN {X 0.051,Y -391.004,Z 1071.608,A 0.000,B 0.000,C 90.000,E1 289.504} C_DIS
LIN {X -0.194,Y -404.754,Z 1071.602,A 0.000,B 0.000,C 90.000,E1 288.362} C_DIS
LIN {X -0.102,Y -415.557,Z 1071.597,A 0.000,B 0.000,C 90.000,E1 287.402} C_DIS
LIN {X -0.116,Y -423.394,Z 1071.593,A 0.000,B 0.000,C 90.000,E1 286.677} C_DIS
LIN {X 0.116,Y -430.960,Z 1071.588,A 0.000,B 0.000,C 90.000,E1 285.898} C_DIS
LIN {X -0.197,Y -440.789,Z 1071.583,A 0.000,B 0.000,C 90.000,E1 284.898} C_DIS
LIN {X 0.130,Y -447.755,Z 1071.578,A 0.000,B 0.000,C 90.000,E1 284.064} C_DIS
LIN {X -0.028,Y -454.241,Z 1071.574,A 0.000,B 0.000,C 90.000,E1 283.300} C_DIS
LIN {X -0.136,Y -460.065,Z 1071.570,A 0.000,B 0.000,C 90.000,E1 282.535} C_DIS
LIN {X -0.189,Y -465.120,Z 1071.565,A 0.000,B 0.000,C 90.000,E1 281.771} C_DIS
LIN {X 0.255,Y -469.489,Z 1071.561,A 0.000,B 0.000,C 90.000,E1 280.950} C_DIS
LIN {X 0.196,Y -473.199,Z 1071.557,A 0.000,B 0.000,C 90.000,E1 280.197} C_DIS
LIN {X 0.170,Y -476.294,Z 1071.553,A 0.000,B 0.000,C 90.000,E1 279.443} C_DIS
LIN {X -0.101,Y -478.061,Z 1071.550,A 0.000,B 0.000,C 90.000,E1 278.973} C_DIS
LIN {X 0.036,Y -479.577,Z 1071.547,A 0.000,B 0.000,C 90.000,E1 278.454} C_DIS
LIN {X -0.067,Y -482.070,Z 1071.541,A 0.000,B 0.000,C 90.000,E1 277.466} C_DIS
LIN {X 0.099,Y -483.037,Z 1071.539,A 0.000,B 0.000,C 90.000,E1 276.947} C_DIS
LIN {X -0.207,Y -483.784,Z 1071.536,A 0.000,B 0.000,C 90.000,E1 276.486} C_DIS
LIN {X -0.027,Y -484.224,Z 1071.533,A 0.000,B 0.000,C 90.000,E1 275.967} C_DIS
LIN {X 0.110,Y -484.314,Z 1071.530,A 0.000,B 0.000,C 90.000,E1 275.454} C_DIS
LIN {X -0.184,Y -483.994,Z 1071.528,A 0.000,B 0.000,C 90.000,E1 274.992} C_DIS
LIN {X 0.003,Y -483.248,Z 1071.525,A 0.000,B 0.000,C 90.000,E1 274.473} C_DIS
LIN {X 0.185,Y -481.897,Z 1071.522,A 0.000,B 0.000,C 90.000,E1 273.955} C_DIS
LIN {X -0.150,Y -480.003,Z 1071.519,A 0.000,B 0.000,C 90.000,E1 273.498} C_DIS
LIN {X 0.016,Y -477.473,Z 1071.517,A 0.000,B 0.000,C 90.000,E1 272.980} C_DIS
LIN {X 0.138,Y -474.195,Z 1071.514,A 0.000,B 0.000,C 90.000,E1 272.465} C_DIS
LIN {X -0.225,Y -469.980,Z 1071.511,A 0.000,B 0.000,C 90.000,E1 272.007} C_DIS
LIN {X -0.122,Y -464.706,Z 1071.508,A 0.000,B 0.000,C 90.000,E1 271.489} C_DIS
LIN {X -0.225,Y -458.868,Z 1071.506,A 0.000,B 0.000,C 90.000,E1 271.031} C_DIS
LIN {X 0.089,Y -452.536,Z 1071.503,A 0.000,B 0.000,C 90.000,E1 270.573} C_DIS
LIN {X -0.055,Y -445.681,Z 1071.501,A 0.000,B 0.000,C 90.000,E1 270.229} C_DIS
LIN {X -0.140,Y -438.246,Z 1071.500,A 0.000,B 0.000,C 90.000,E1 269.943} C_DIS
LIN {X -0.143,Y -430.563,Z 1071.498,A 0.000,B 0.000,C 90.000,E1 269.714} C_DIS
LIN {X -0.145,Y -422.578,Z 1071.497,A 0.000,B 0.000,C 90.000,E1 269.542} C_DIS
LIN {X 0.176,Y -413.717,Z 1071.497,A 0.000,B 0.000,C 90.000,E1 269.370} C_DIS
LIN {X -0.184,Y -401.939,Z 1071.496,A 0.000,B 0.000,C 90.000,E1 269.312} C_DIS
LIN {X 0.024,Y -394.839,Z 1071.496,A 0.000,B 0.000,C 90.000,E1 269.255} C_DIS
LIN {X -0.017,Y -181.377,Z 1071.496,A 0.000,B 0.000,C 90.000,E1 269.255} C_DIS
LIN {X 0.013,Y -180.907,Z 1071.475,A 0.000,B 0.000,C 90.000,E1 265.527} C_DIS
LIN {X 0.070,Y -180.762,Z 1071.470,A 0.000,B 0.000,C 90.000,E1 264.666} C_DIS
LIN {X -0.038,Y -178.856,Z 1071.442,A 0.000,B 0.000,C 90.000,E1 259.634} C_DIS
LIN {X 0.033,Y -175.899,Z 1071.414,A 0.000,B 0.000,C 90.000,E1 254.519} C_DIS
LIN {X -0.028,Y -174.578,Z 1071.405,A 0.000,B 0.000,C 90.000,E1 252.834} C_DIS
LIN {X 0.007,Y -171.561,Z 1071.381,A 0.000,B 0.000,C 90.000,E1 248.539} C_DIS
LIN {X -0.010,Y -167.785,Z 1071.357,A 0.000,B 0.000,C 90.000,E1 244.229} C_DIS
LIN {X 0.004,Y -166.498,Z 1071.347,A 0.000,B 0.000,C 90.000,E1 242.487} C_DIS
LIN {X 0.000,Y -163.208,Z 1071.328,A 0.000,B 0.000,C 90.000,E1 238.997} C_DIS
LIN {X -0.035,Y -161.172,Z 1071.313,A 0.000,B 0.000,C 90.000,E1 236.373} C_DIS
LIN {X 0.088,Y -157.187,Z 1071.289,A 0.000,B 0.000,C 90.000,E1 231.904} C_DIS
LIN {X 0.011,Y -155.917,Z 1071.279,A 0.000,B 0.000,C 90.000,E1 230.150} C_DIS
LIN {X 0.067,Y -152.167,Z 1071.254,A 0.000,B 0.000,C 90.000,E1 225.648} C_DIS
LIN {X -0.023,Y -150.416,Z 1071.239,A 0.000,B 0.000,C 90.000,E1 222.975} C_DIS
LIN {X 0.018,Y -147.144,Z 1071.214,A 0.000,B 0.000,C 90.000,E1 218.418} C_DIS
LIN {X 0.015,Y -145.702,Z 1071.198,A 0.000,B 0.000,C 90.000,E1 215.678} C_DIS
LIN {X 0.023,Y -143.085,Z 1071.173,A 0.000,B 0.000,C 90.000,E1 211.082} C_DIS
LIN {X 0.028,Y -141.702,Z 1071.152,A 0.000,B 0.000,C 90.000,E1 207.385} C_DIS
LIN {X -0.049,Y -139.468,Z 1071.116,A 0.000,B 0.000,C 90.000,E1 200.918} C_DIS
LIN {X 0.004,Y -139.200,Z 1071.106,A 0.000,B 0.000,C 90.000,E1 199.033} C_DIS
LIN {X 0.068,Y -138.328,Z 1071.054,A 0.000,B 0.000,C 90.000,E1 189.670} C_DIS
LIN {X -0.066,Y -139.444,Z 1071.007,A 0.000,B 0.000,C 90.000,E1 181.318} C_DIS
LIN {X 0.014,Y -140.981,Z 1070.976,A 0.000,B 0.000,C 90.000,E1 175.698} C_DIS
LIN {X -0.037,Y -142.737,Z 1070.956,A 0.000,B 0.000,C 90.000,E1 172.008} C_DIS
LIN {X 0.062,Y -145.127,Z 1070.930,A 0.000,B 0.000,C 90.000,E1 167.353} C_DIS
LIN {X 0.055,Y -147.750,Z 1070.909,A 0.000,B 0.000,C 90.000,E1 163.685} C_DIS
LIN {X -0.006,Y -150.419,Z 1070.889,A 0.000,B 0.000,C 90.000,E1 160.061} C_DIS
LIN {X 0.010,Y -153.859,Z 1070.869,A 0.000,B 0.000,C 90.000,E1 156.433} C_DIS
LIN {X -0.073,Y -157.270,Z 1070.849,A 0.000,B 0.000,C 90.000,E1 152.871} C_DIS
LIN {X 0.005,Y -161.447,Z 1070.829,A 0.000,B 0.000,C 90.000,E1 149.282} C_DIS
LIN {X 0.011,Y -165.648,Z 1070.810,A 0.000,B 0.000,C 90.000,E1 145.754} C_DIS
LIN {X -0.007,Y -170.582,Z 1070.790,A 0.000,B 0.000,C 90.000,E1 142.271} C_DIS
LIN {X -0.100,Y -175.459,Z 1070.771,A 0.000,B 0.000,C 90.000,E1 138.852} C_DIS
LIN {X 0.016,Y -181.083,Z 1070.752,A 0.000,B 0.000,C 90.000,E1 135.405} C_DIS
LIN {X 0.005,Y -186.523,Z 1070.734,A 0.000,B 0.000,C 90.000,E1 132.043} C_DIS
LIN {X -0.053,Y -191.140,Z 1070.720,A 0.000,B 0.000,C 90.000,E1 129.564} C_DIS
LIN {X 0.026,Y -196.941,Z 1070.701,A 0.000,B 0.000,C 90.000,E1 126.251} C_DIS
LIN {X 0.053,Y -198.936,Z 1070.696,A 0.000,B 0.000,C 90.000,E1 125.231} C_DIS
LIN {X 0.045,Y -305.778,Z 1070.696,A 0.000,B 0.000,C 90.000,E1 125.231} C_DIS
LIN {X -0.005,Y -308.437,Z 1070.695,A 0.000,B 0.000,C 90.000,E1 125.185} C_DIS
LIN {X 0.047,Y -313.253,Z 1070.694,A 0.000,B 0.000,C 90.000,E1 124.898} C_DIS
LIN {X 0.098,Y -316.007,Z 1070.692,A 0.000,B 0.000,C 90.000,E1 124.612} C_DIS
LIN {X -0.030,Y -319.686,Z 1070.689,A 0.000,B 0.000,C 90.000,E1 124.072} C_DIS
LIN {X 0.217,Y -321.153,Z 1070.688,A 0.000,B 0.000,C 90.000,E1 123.706} C_DIS
LIN {X 0.026,Y -333.881,Z 1070.668,A 0.000,B 0.000,C 90.000,E1 120.256} C_DIS
LIN {X 0.048,Y -345.712,Z 1070.653,A 0.000,B 0.000,C 90.000,E1 117.462} C_DIS
LIN {X 0.102,Y -359.001,Z 1070.637,A 0.000,B 0.000,C 90.000,E1 114.719} C_DIS
LIN {X 0.145,Y -372.129,Z 1070.624,A 0.000,B 0.000,C 90.000,E1 112.333} C_DIS
LIN {X 0.228,Y -386.591,Z 1070.611,A 0.000,B 0.000,C 90.000,E1 109.993} C_DIS
LIN {X -0.091,Y -402.491,Z 1070.599,A 0.000,B 0.000,C 90.000,E1 107.764} C_DIS
LIN {X -0.145,Y -419.941,Z 1070.586,A 0.000,B 0.000,C 90.000,E1 105.552} C_DIS
LIN {X 0.132,Y -439.051,Z 1070.574,A 0.000,B 0.000,C 90.000,E1 103.355} C_DIS
LIN {X -0.115,Y -459.150,Z 1070.563,A 0.000,B 0.000,C 90.000,E1 101.366} C_DIS
LIN {X -0.160,Y -466.817,Z 1070.559,A 0.000,B 0.000,C 90.000,E1 100.658} C_DIS
LIN {X -0.149,Y -469.091,Z 1070.558,A 0.000,B 0.000,C 90.000,E1 100.423} C_DIS
LIN {X 0.095,Y -470.915,Z 1070.556,A 0.000,B 0.000,C 90.000,E1 100.141} C_DIS
LIN {X -0.042,Y -472.288,Z 1070.555,A 0.000,B 0.000,C 90.000,E1 99.905} C_DIS
LIN {X 0.139,Y -474.035,Z 1070.552,A 0.000,B 0.000,C 90.000,E1 99.378} C_DIS
LIN {X -0.219,Y -474.702,Z 1070.549,A 0.000,B 0.000,C 90.000,E1 98.916} C_DIS
LIN {X -0.095,Y -474.401,Z 1070.547,A 0.000,B 0.000,C 90.000,E1 98.398} C_DIS
LIN {X 0.100,Y -473.094,Z 1070.544,A 0.000,B 0.000,C 90.000,E1 97.871} C_DIS
LIN {X -0.104,Y -471.998,Z 1070.542,A 0.000,B 0.000,C 90.000,E1 97.644} C_DIS
LIN {X 0.224,Y -470.534,Z 1070.541,A 0.000,B 0.000,C 90.000,E1 97.352} C_DIS
LIN {X 0.087,Y -456.259,Z 1070.530,A 0.000,B 0.000,C 90.000,E1 95.334} C_DIS
LIN {X 0.010,Y -442.027,Z 1070.518,A 0.000,B 0.000,C 90.000,E1 93.269} C_DIS
LIN {X 0.037,Y -424.226,Z 1070.502,A 0.000,B 0.000,C 90.000,E1 90.344} C_DIS
LIN {X -0.011,Y -406.215,Z 1070.484,A 0.000,B 0.000,C 90.000,E1 87.078} C_DIS
LIN {X -0.042,Y -397.225,Z 1070.474,A 0.000,B 0.000,C 90.000,E1 85.412} C_DIS
LIN {X -0.193,Y -388.040,Z 1070.465,A 0.000,B 0.000,C 90.000,E1 83.742} C_DIS
LIN {X -0.105,Y -377.106,Z 1070.454,A 0.000,B 0.000,C 90.000,E1 81.724} C_DIS
LIN {X -0.134,Y -367.469,Z 1070.444,A 0.000,B 0.000,C 90.000,E1 79.982} C_DIS
LIN {X 0.083,Y -357.534,Z 1070.434,A 0.000,B 0.000,C 90.000,E1 78.173} C_DIS
LIN {X 0.112,Y -345.875,Z 1070.423,A 0.000,B 0.000,C 90.000,E1 76.061} C_DIS
LIN {X 0.045,Y -332.783,Z 1070.409,A 0.000,B 0.000,C 90.000,E1 73.614} C_DIS
LIN {X 0.030,Y -318.650,Z 1070.393,A 0.000,B 0.000,C 90.000,E1 70.786} C_DIS
LIN {X -0.052,Y -305.252,Z 1070.377,A 0.000,B 0.000,C 90.000,E1 67.901} C_DIS
LIN {X -0.128,Y -295.264,Z 1070.364,A 0.000,B 0.000,C 90.000,E1 65.613} C_DIS
LIN {X -0.065,Y -285.408,Z 1070.351,A 0.000,B 0.000,C 90.000,E1 63.256} C_DIS
LIN {X -0.006,Y -274.402,Z 1070.336,A 0.000,B 0.000,C 90.000,E1 60.511} C_DIS
LIN {X 0.052,Y -263.635,Z 1070.321,A 0.000,B 0.000,C 90.000,E1 57.709} C_DIS
LIN {X -0.098,Y -253.284,Z 1070.305,A 0.000,B 0.000,C 90.000,E1 54.895} C_DIS
LIN {X -0.070,Y -243.326,Z 1070.289,A 0.000,B 0.000,C 90.000,E1 51.984} C_DIS
LIN {X 0.089,Y -232.766,Z 1070.270,A 0.000,B 0.000,C 90.000,E1 48.609} C_DIS
LIN {X -0.004,Y -223.972,Z 1070.253,A 0.000,B 0.000,C 90.000,E1 45.607} C_DIS
LIN {X 0.014,Y -215.696,Z 1070.236,A 0.000,B 0.000,C 90.000,E1 42.528} C_DIS
LIN {X 0.002,Y -207.798,Z 1070.219,A 0.000,B 0.000,C 90.000,E1 39.402} C_DIS
LIN {X 0.014,Y -200.480,Z 1070.201,A 0.000,B 0.000,C 90.000,E1 36.217} C_DIS
LIN {X 0.099,Y -193.737,Z 1070.183,A 0.000,B 0.000,C 90.000,E1 32.959} C_DIS
LIN {X -0.029,Y -187.770,Z 1070.165,A 0.000,B 0.000,C 90.000,E1 29.716} C_DIS
LIN {X 0.073,Y -182.459,Z 1070.147,A 0.000,B 0.000,C 90.000,E1 26.360} C_DIS
LIN {X -0.021,Y -177.915,Z 1070.128,A 0.000,B 0.000,C 90.000,E1 23.025} C_DIS
LIN {X -0.033,Y -174.021,Z 1070.109,A 0.000,B 0.000,C 90.000,E1 19.631} C_DIS
LIN {X 0.039,Y -170.183,Z 1070.085,A 0.000,B 0.000,C 90.000,E1 15.315} C_DIS
LIN {X -0.015,Y -167.361,Z 1070.061,A 0.000,B 0.000,C 90.000,E1 11.007} C_DIS
LIN {X 0.064,Y -165.103,Z 1070.027,A 0.000,B 0.000,C 90.000,E1 4.878} C_DIS
LIN {X -0.007,Y -166.278,Z 1069.958,A 0.000,B 0.000,C 90.000,E1 352.534} C_DIS
LIN {X 0.025,Y -169.162,Z 1069.929,A 0.000,B 0.000,C 90.000,E1 347.297} C_DIS
LIN {X 0.062,Y -172.764,Z 1069.905,A 0.000,B 0.000,C 90.000,E1 342.960} C_DIS
LIN {X -0.072,Y -176.344,Z 1069.886,A 0.000,B 0.000,C 90.000,E1 339.571} C_DIS
LIN {X -0.102,Y -180.678,Z 1069.867,A 0.000,B 0.000,C 90.000,E1 336.177} C_DIS
LIN {X -0.059,Y -185.671,Z 1069.849,A 0.000,B 0.000,C 90.000,E1 332.794} C_DIS
LIN {X -0.043,Y -191.538,Z 1069.830,A 0.000,B 0.000,C 90.000,E1 329.459} C_DIS
LIN {X -0.021,Y -198.235,Z 1069.812,A 0.000,B 0.000,C 90.000,E1 326.167} C_DIS
LIN {X 0.002,Y -205.625,Z 1069.794,A 0.000,B 0.000,C 90.000,E1 322.924} C_DIS
LIN {X -0.098,Y -214.828,Z 1069.774,A 0.000,B 0.000,C 90.000,E1 319.380} C_DIS
LIN {X 0.097,Y -223.687,Z 1069.757,A 0.000,B 0.000,C 90.000,E1 316.215} C_DIS
LIN {X 0.040,Y -233.437,Z 1069.740,A 0.000,B 0.000,C 90.000,E1 313.176} C_DIS
LIN {X 0.092,Y -244.621,Z 1069.723,A 0.000,B 0.000,C 90.000,E1 310.172} C_DIS
LIN {X -0.107,Y -252.562,Z 1069.713,A 0.000,B 0.000,C 90.000,E1 308.382} C_DIS
LIN {X -0.054,Y -265.032,Z 1069.699,A 0.000,B 0.000,C 90.000,E1 305.851} C_DIS
LIN {X 0.075,Y -282.586,Z 1069.682,A 0.000,B 0.000,C 90.000,E1 302.673} C_DIS
LIN {X -0.119,Y -301.555,Z 1069.665,A 0.000,B 0.000,C 90.000,E1 299.667} C_DIS
LIN {X 0.056,Y -322.064,Z 1069.648,A 0.000,B 0.000,C 90.000,E1 296.693} C_DIS
LIN {X 0.074,Y -334.438,Z 1069.640,A 0.000,B 0.000,C 90.000,E1 295.103} C_DIS
LIN {X 0.058,Y -347.744,Z 1069.631,A 0.000,B 0.000,C 90.000,E1 293.590} C_DIS
LIN {X -0.006,Y -363.800,Z 1069.622,A 0.000,B 0.000,C 90.000,E1 291.972} C_DIS
LIN {X -0.169,Y -388.553,Z 1069.610,A 0.000,B 0.000,C 90.000,E1 289.758} C_DIS
LIN {X 0.024,Y -405.070,Z 1069.602,A 0.000,B 0.000,C 90.000,E1 288.308} C_DIS
LIN {X -0.195,Y -413.085,Z 1069.598,A 0.000,B 0.000,C 90.000,E1 287.638} C_DIS
LIN {X -0.137,Y -423.457,Z 1069.593,A 0.000,B 0.000,C 90.000,E1 286.677} C_DIS
LIN {X 0.130,Y -430.955,Z 1069.588,A 0.000,B 0.000,C 90.000,E1 285.898} C_DIS
LIN {X -0.187,Y -440.766,Z 1069.583,A 0.000,B 0.000,C 90.000,E1 284.898} C_DIS
LIN {X 0.136,Y -447.735,Z 1069.578,A 0.000,B 0.000,C 90.000,E1 284.064} C_DIS
LIN {X -0.022,Y -454.225,Z 1069.574,A 0.000,B 0.000,C 90.000,E1 283.300} C_DIS
LIN {X -0.130,Y -460.077,Z 1069.570,A 0.000,B 0.000,C 90.000,E1 282.535} C_DIS
LIN {X -0.183,Y -465.167,Z 1069.565,A 0.000,B 0.000,C 90.000,E1 281.771} C_DIS
LIN {X -0.200,Y -469.551,Z 1069.561,A 0.000,B 0.000,C 90.000,E1 281.007} C_DIS
LIN {X 0.203,Y -473.261,Z 1069.557,A 0.000,B 0.000,C 90.000,E1 280.197} C_DIS
LIN {X 0.177,Y -476.396,Z 1069.553,A 0.000,B 0.000,C 90.000,E1 279.443} C_DIS
LIN {X -0.093,Y -478.179,Z 1069.550,A 0.000,B 0.000,C 90.000,E1 278.973} C_DIS
LIN {X 0.044,Y -479.711,Z 1069.547,A 0.000,B 0.000,C 90.000,E1 278.454} C_DIS
LIN {X -0.057,Y -482.226,Z 1069.541,A 0.000,B 0.000,C 90.000,E1 277.466} C_DIS
LIN {X 0.110,Y -483.221,Z 1069.539,A 0.000,B 0.000,C 90.000,E1 276.947} C_DIS
LIN {X -0.196,Y -484.003,Z 1069.536,A 0.000,B 0.000,C 90.000,E1 276.486} C_DIS
LIN {X -0.015,Y -484.467,Z 1069.533,A 0.000,B 0.000,C 90.000,E1 275.967} C_DIS
LIN {X 0.123,Y -484.574,Z 1069.530,A 0.000,B 0.000,C 90.000,E1 275.454} C_DIS
LIN {X -0.169,Y -484.257,Z 1069.528,A 0.000,B 0.000,C 90.000,E1 274.992} C_DIS
LIN {X 0.020,Y -483.494,Z 1069.525,A 0.000,B 0.000,C 90.000,E1 274.473} C_DIS
LIN {X 0.203,Y -482.209,Z 1069.522,A 0.000,B 0.000,C 90.000,E1 273.955} C_DIS
LIN {X 0.179,Y -479.151,Z 1069.518,A 0.000,B 0.000,C 90.000,E1 273.212} C_DIS
LIN {X -0.139,Y -476.226,Z 1069.515,A 0.000,B 0.000,C 90.000,E1 272.751} C_DIS
LIN {X -0.021,Y -472.477,Z 1069.512,A 0.000,B 0.000,C 90.000,E1 272.236} C_DIS
LIN {X -0.201,Y -470.291,Z 1069.511,A 0.000,B 0.000,C 90.000,E1 272.007} C_DIS
LIN {X -0.097,Y -465.064,Z 1069.508,A 0.000,B 0.000,C 90.000,E1 271.489} C_DIS
LIN {X -0.208,Y -459.236,Z 1069.506,A 0.000,B 0.000,C 90.000,E1 271.031} C_DIS
LIN {X 0.088,Y -452.905,Z 1069.503,A 0.000,B 0.000,C 90.000,E1 270.573} C_DIS
LIN {X -0.065,Y -446.126,Z 1069.501,A 0.000,B 0.000,C 90.000,E1 270.229} C_DIS
LIN {X -0.169,Y -438.712,Z 1069.500,A 0.000,B 0.000,C 90.000,E1 269.943} C_DIS
LIN {X -0.183,Y -431.085,Z 1069.498,A 0.000,B 0.000,C 90.000,E1 269.714} C_DIS
LIN {X -0.197,Y -423.165,Z 1069.497,A 0.000,B 0.000,C 90.000,E1 269.542} C_DIS
LIN {X 0.126,Y -414.412,Z 1069.497,A 0.000,B 0.000,C 90.000,E1 269.370} C_DIS
LIN {X -0.116,Y -405.428,Z 1069.496,A 0.000,B 0.000,C 90.000,E1 269.312} C_DIS
LIN {X -0.041,Y -396.553,Z 1069.496,A 0.000,B 0.000,C 90.000,E1 269.255} C_DIS
LIN {X -0.105,Y -391.286,Z 1069.496,A 0.000,B 0.000,C 90.000,E1 269.255} C_DIS
LIN {X -0.078,Y -181.372,Z 1069.496,A 0.000,B 0.000,C 90.000,E1 269.255} C_DIS
LIN {X -0.020,Y -180.908,Z 1069.475,A 0.000,B 0.000,C 90.000,E1 265.527} C_DIS
LIN {X 0.037,Y -180.758,Z 1069.470,A 0.000,B 0.000,C 90.000,E1 264.666} C_DIS
LIN {X -0.071,Y -178.851,Z 1069.442,A 0.000,B 0.000,C 90.000,E1 259.634} C_DIS
LIN {X 0.000,Y -175.895,Z 1069.414,A 0.000,B 0.000,C 90.000,E1 254.519} C_DIS
LIN {X -0.060,Y -174.569,Z 1069.405,A 0.000,B 0.000,C 90.000,E1 252.834} C_DIS
LIN {X -0.025,Y -171.553,Z 1069.381,A 0.000,B 0.000,C 90.000,E1 248.539} C_DIS
LIN {X 0.031,Y -167.777,Z 1069.357,A 0.000,B 0.000,C 90.000,E1 244.204} C_DIS
LIN {X -0.027,Y -166.488,Z 1069.347,A 0.000,B 0.000,C 90.000,E1 242.487} C_DIS
LIN {X -0.031,Y -163.199,Z 1069.328,A 0.000,B 0.000,C 90.000,E1 238.997} C_DIS
LIN {X 0.023,Y -161.163,Z 1069.313,A 0.000,B 0.000,C 90.000,E1 236.342} C_DIS
LIN {X 0.059,Y -157.178,Z 1069.288,A 0.000,B 0.000,C 90.000,E1 231.904} C_DIS
LIN {X -0.019,Y -155.909,Z 1069.279,A 0.000,B 0.000,C 90.000,E1 230.150} C_DIS
LIN {X 0.038,Y -152.159,Z 1069.254,A 0.000,B 0.000,C 90.000,E1 225.648} C_DIS
LIN {X 0.058,Y -150.408,Z 1069.239,A 0.000,B 0.000,C 90.000,E1 222.933} C_DIS
LIN {X 0.081,Y -147.137,Z 1069.213,A 0.000,B 0.000,C 90.000,E1 218.382} C_DIS
LIN {X -0.014,Y -145.698,Z 1069.198,A 0.000,B 0.000,C 90.000,E1 215.678} C_DIS
LIN {X -0.005,Y -143.080,Z 1069.173,A 0.000,B 0.000,C 90.000,E1 211.082} C_DIS
LIN {X -0.001,Y -141.699,Z 1069.152,A 0.000,B 0.000,C 90.000,E1 207.385} C_DIS
LIN {X -0.077,Y -139.465,Z 1069.116,A 0.000,B 0.000,C 90.000,E1 200.918} C_DIS
LIN {X -0.024,Y -139.198,Z 1069.106,A 0.000,B 0.000,C 90.000,E1 199.033} C_DIS
LIN {X 0.040,Y -138.327,Z 1069.054,A 0.000,B 0.000,C 90.000,E1 189.670} C_DIS
LIN {X 0.045,Y -139.447,Z 1069.007,A 0.000,B 0.000,C 90.000,E1 181.260} C_DIS
LIN {X -0.015,Y -140.985,Z 1068.976,A 0.000,B 0.000,C 90.000,E1 175.698} C_DIS
LIN {X -0.065,Y -142.741,Z 1068.955,A 0.000,B 0.000,C 90.000,E1 172.008} C_DIS
LIN {X 0.033,Y -145.134,Z 1068.930,A 0.000,B 0.000,C 90.000,E1 167.353} C_DIS
LIN {X 0.026,Y -147.758,Z 1068.909,A 0.000,B 0.000,C 90.000,E1 163.685} C_DIS
LIN {X -0.035,Y -150.428,Z 1068.889,A 0.000,B 0.000,C 90.000,E1 160.061} C_DIS
LIN {X -0.020,Y -153.871,Z 1068.869,A 0.000,B 0.000,C 90.000,E1 156.433} C_DIS
LIN {X 0.037,Y -157.282,Z 1068.849,A 0.000,B 0.000,C 90.000,E1 152.820} C_DIS
LIN {X -0.026,Y -161.462,Z 1068.829,A 0.000,B 0.000,C 90.000,E1 149.282} C_DIS
LIN {X -0.020,Y -165.662,Z 1068.810,A 0.000,B 0.000,C 90.000,E1 145.754} C_DIS
LIN {X -0.038,Y -170.599,Z 1068.790,A 0.000,B 0.000,C 90.000,E1 142.271} C_DIS
LIN {X 0.000,Y -175.476,Z 1068.771,A 0.000,B 0.000,C 90.000,E1 138.809} C_DIS
LIN {X -0.017,Y -181.098,Z 1068.752,A 0.000,B 0.000,C 90.000,E1 135.405} C_DIS
LIN {X -0.028,Y -186.541,Z 1068.734,A 0.000,B 0.000,C 90.000,E1 132.043} C_DIS
LIN {X -0.086,Y -191.158,Z 1068.720,A 0.000,B 0.000,C 90.000,E1 129.564} C_DIS
LIN {X -0.009,Y -196.960,Z 1068.701,A 0.000,B 0.000,C 90.000,E1 126.251} C_DIS
LIN {X -0.083,Y -198.853,Z 1068.696,A 0.000,B 0.000,C 90.000,E1 125.311} C_DIS
LIN {X -0.162,Y -305.870,Z 1068.696,A 0.000,B 0.000,C 90.000,E1 125.311} C_DIS
LIN {X 0.029,Y -307.987,Z 1068.696,A 0.000,B 0.000,C 90.000,E1 125.231} C_DIS
LIN {X -0.093,Y -313.359,Z 1068.694,A 0.000,B 0.000,C 90.000,E1 124.945} C_DIS
LIN {X 0.043,Y -316.285,Z 1068.692,A 0.000,B 0.000,C 90.000,E1 124.612} C_DIS
LIN {X 0.011,Y -318.306,Z 1068.691,A 0.000,B 0.000,C 90.000,E1 124.326} C_DIS
LIN {X -0.022,Y -319.892,Z 1068.689,A 0.000,B 0.000,C 90.000,E1 124.040} C_DIS
LIN {X 0.052,Y -321.273,Z 1068.687,A 0.000,B 0.000,C 90.000,E1 123.706} C_DIS
LIN {X 0.034,Y -332.735,Z 1068.670,A 0.000,B 0.000,C 90.000,E1 120.541} C_DIS
LIN {X -0.115,Y -344.428,Z 1068.654,A 0.000,B 0.000,C 90.000,E1 117.769} C_DIS
LIN {X -0.108,Y -357.561,Z 1068.639,A 0.000,B 0.000,C 90.000,E1 115.027} C_DIS
LIN {X -0.112,Y -370.542,Z 1068.626,A 0.000,B 0.000,C 90.000,E1 112.642} C_DIS
LIN {X -0.078,Y -384.847,Z 1068.613,A 0.000,B 0.000,C 90.000,E1 110.301} C_DIS
LIN {X 0.055,Y -400.577,Z 1068.600,A 0.000,B 0.000,C 90.000,E1 108.000} C_DIS
LIN {X -0.044,Y -417.843,Z 1068.588,A 0.000,B 0.000,C 90.000,E1 105.788} C_DIS
LIN {X 0.181,Y -436.762,Z 1068.576,A 0.000,B 0.000,C 90.000,E1 103.592} C_DIS
LIN {X -0.131,Y -456.793,Z 1068.564,A 0.000,B 0.000,C 90.000,E1 101.591} C_DIS
LIN {X 0.127,Y -467.020,Z 1068.559,A 0.000,B 0.000,C 90.000,E1 100.602} C_DIS
LIN {X 0.140,Y -469.236,Z 1068.558,A 0.000,B 0.000,C 90.000,E1 100.366} C_DIS
LIN {X -0.095,Y -471.032,Z 1068.556,A 0.000,B 0.000,C 90.000,E1 100.141} C_DIS
LIN {X -0.248,Y -472.380,Z 1068.555,A 0.000,B 0.000,C 90.000,E1 99.905} C_DIS
LIN {X -0.068,Y -474.069,Z 1068.552,A 0.000,B 0.000,C 90.000,E1 99.378} C_DIS
LIN {X 0.044,Y -474.689,Z 1068.549,A 0.000,B 0.000,C 90.000,E1 98.859} C_DIS
LIN {X 0.169,Y -474.344,Z 1068.547,A 0.000,B 0.000,C 90.000,E1 98.341} C_DIS
LIN {X -0.105,Y -472.985,Z 1068.544,A 0.000,B 0.000,C 90.000,E1 97.871} C_DIS
LIN {X 0.160,Y -471.857,Z 1068.542,A 0.000,B 0.000,C 90.000,E1 97.587} C_DIS
LIN {X 0.020,Y -470.354,Z 1068.541,A 0.000,B 0.000,C 90.000,E1 97.352} C_DIS
LIN {X -0.114,Y -456.061,Z 1068.530,A 0.000,B 0.000,C 90.000,E1 95.334} C_DIS
LIN {X -0.190,Y -441.841,Z 1068.518,A 0.000,B 0.000,C 90.000,E1 93.269} C_DIS
LIN {X -0.160,Y -424.056,Z 1068.502,A 0.000,B 0.000,C 90.000,E1 90.344} C_DIS
LIN {X 0.132,Y -407.557,Z 1068.485,A 0.000,B 0.000,C 90.000,E1 87.306} C_DIS
LIN {X 0.125,Y -398.599,Z 1068.476,A 0.000,B 0.000,C 90.000,E1 85.641} C_DIS
LIN {X -0.002,Y -389.437,Z 1068.467,A 0.000,B 0.000,C 90.000,E1 83.970} C_DIS
LIN {X 0.112,Y -378.550,Z 1068.455,A 0.000,B 0.000,C 90.000,E1 81.951} C_DIS
LIN {X 0.109,Y -368.931,Z 1068.446,A 0.000,B 0.000,C 90.000,E1 80.208} C_DIS
LIN {X -0.068,Y -359.030,Z 1068.436,A 0.000,B 0.000,C 90.000,E1 78.465} C_DIS
LIN {X -0.071,Y -345.687,Z 1068.422,A 0.000,B 0.000,C 90.000,E1 76.061} C_DIS
LIN {X 0.184,Y -332.618,Z 1068.409,A 0.000,B 0.000,C 90.000,E1 73.559} C_DIS
LIN {X 0.155,Y -318.494,Z 1068.393,A 0.000,B 0.000,C 90.000,E1 70.732} C_DIS
LIN {X -0.035,Y -303.662,Z 1068.375,A 0.000,B 0.000,C 90.000,E1 67.539} C_DIS
LIN {X -0.036,Y -293.670,Z 1068.362,A 0.000,B 0.000,C 90.000,E1 65.229} C_DIS
LIN {X -0.004,Y -283.822,Z 1068.349,A 0.000,B 0.000,C 90.000,E1 62.871} C_DIS
LIN {X 0.012,Y -272.877,Z 1068.334,A 0.000,B 0.000,C 90.000,E1 60.127} C_DIS
LIN {X 0.074,Y -260.819,Z 1068.317,A 0.000,B 0.000,C 90.000,E1 56.962} C_DIS
LIN {X -0.003,Y -250.507,Z 1068.301,A 0.000,B 0.000,C 90.000,E1 54.116} C_DIS
LIN {X 0.092,Y -239.461,Z 1068.282,A 0.000,B 0.000,C 90.000,E1 50.803} C_DIS
LIN {X -0.041,Y -229.123,Z 1068.264,A 0.000,B 0.000,C 90.000,E1 47.472} C_DIS
LIN {X 0.023,Y -219.509,Z 1068.245,A 0.000,B 0.000,C 90.000,E1 44.028} C_DIS
LIN {X 0.089,Y -211.433,Z 1068.227,A 0.000,B 0.000,C 90.000,E1 40.906} C_DIS
LIN {X -0.133,Y -203.794,Z 1068.210,A 0.000,B 0.000,C 90.000,E1 37.810} C_DIS
LIN {X 0.105,Y -196.764,Z 1068.192,A 0.000,B 0.000,C 90.000,E1 34.532} C_DIS
LIN {X -0.111,Y -190.409,Z 1068.174,A 0.000,B 0.000,C 90.000,E1 31.337} C_DIS
LIN {X 0.077,Y -184.778,Z 1068.156,A 0.000,B 0.000,C 90.000,E1 27.975} C_DIS
LIN {X 0.027,Y -179.856,Z 1068.137,A 0.000,B 0.000,C 90.000,E1 24.643} C_DIS
LIN {X -0.039,Y -175.627,Z 1068.118,A 0.000,B 0.000,C 90.000,E1 21.280} C_DIS
LIN {X -0.068,Y -172.134,Z 1068.099,A 0.000,B 0.000,C 90.000,E1 17.873} C_DIS
LIN {X 0.018,Y -168.721,Z 1068.075,A 0.000,B 0.000,C 90.000,E1 13.536} C_DIS
LIN {X -0.035,Y -166.004,Z 1068.046,A 0.000,B 0.000,C 90.000,E1 8.341} C_DIS
LIN {X -0.011,Y -166.500,Z 1067.954,A 0.000,B 0.000,C 90.000,E1 351.659} C_DIS
LIN {X 0.011,Y -169.002,Z 1067.929,A 0.000,B 0.000,C 90.000,E1 347.297} C_DIS
LIN {X 0.042,Y -172.608,Z 1067.905,A 0.000,B 0.000,C 90.000,E1 342.960} C_DIS
LIN {X 0.070,Y -176.183,Z 1067.886,A 0.000,B 0.000,C 90.000,E1 339.518} C_DIS
LIN {X 0.034,Y -180.531,Z 1067.867,A 0.000,B 0.000,C 90.000,E1 336.125} C_DIS
LIN {X 0.073,Y -185.528,Z 1067.849,A 0.000,B 0.000,C 90.000,E1 332.743} C_DIS
LIN {X 0.084,Y -191.421,Z 1067.830,A 0.000,B 0.000,C 90.000,E1 329.410} C_DIS
LIN {X 0.047,Y -198.124,Z 1067.812,A 0.000,B 0.000,C 90.000,E1 326.135} C_DIS
LIN {X 0.124,Y -206.497,Z 1067.792,A 0.000,B 0.000,C 90.000,E1 322.477} C_DIS
LIN {X 0.055,Y -215.789,Z 1067.772,A 0.000,B 0.000,C 90.000,E1 318.933} C_DIS
LIN {X 0.117,Y -224.745,Z 1067.755,A 0.000,B 0.000,C 90.000,E1 315.810} C_DIS
LIN {X 0.028,Y -232.028,Z 1067.742,A 0.000,B 0.000,C 90.000,E1 313.542} C_DIS
LIN {X 0.037,Y -243.031,Z 1067.725,A 0.000,B 0.000,C 90.000,E1 310.539} C_DIS
LIN {X 0.012,Y -250.775,Z 1067.715,A 0.000,B 0.000,C 90.000,E1 308.705} C_DIS
LIN {X -0.007,Y -261.196,Z 1067.703,A 0.000,B 0.000,C 90.000,E1 306.537} C_DIS
LIN {X 0.020,Y -276.500,Z 1067.687,A 0.000,B 0.000,C 90.000,E1 303.706} C_DIS
LIN {X 0.048,Y -295.084,Z 1067.670,A 0.000,B 0.000,C 90.000,E1 300.620} C_DIS
LIN {X 0.073,Y -315.045,Z 1067.654,A 0.000,B 0.000,C 90.000,E1 297.641} C_DIS
LIN {X 0.058,Y -329.397,Z 1067.643,A 0.000,B 0.000,C 90.000,E1 295.720} C_DIS
LIN {X 0.084,Y -339.770,Z 1067.636,A 0.000,B 0.000,C 90.000,E1 294.463} C_DIS
LIN {X -0.042,Y -353.244,Z 1067.628,A 0.000,B 0.000,C 90.000,E1 293.025} C_DIS
LIN {X -0.038,Y -372.631,Z 1067.617,A 0.000,B 0.000,C 90.000,E1 291.153} C_DIS
LIN {X -0.067,Y -391.975,Z 1067.608,A 0.000,B 0.000,C 90.000,E1 289.450} C_DIS
LIN {X 0.167,Y -405.717,Z 1067.601,A 0.000,B 0.000,C 90.000,E1 288.236} C_DIS
LIN {X -0.240,Y -413.796,Z 1067.598,A 0.000,B 0.000,C 90.000,E1 287.583} C_DIS
LIN {X 0.049,Y -424.331,Z 1067.592,A 0.000,B 0.000,C 90.000,E1 286.567} C_DIS
LIN {X -0.183,Y -431.901,Z 1067.588,A 0.000,B 0.000,C 90.000,E1 285.843} C_DIS
LIN {X 0.222,Y -439.249,Z 1067.583,A 0.000,B 0.000,C 90.000,E1 285.009} C_DIS
LIN {X -0.008,Y -446.330,Z 1067.579,A 0.000,B 0.000,C 90.000,E1 284.245} C_DIS
LIN {X -0.079,Y -452.935,Z 1067.575,A 0.000,B 0.000,C 90.000,E1 283.467} C_DIS
LIN {X 0.250,Y -458.880,Z 1067.570,A 0.000,B 0.000,C 90.000,E1 282.647} C_DIS
LIN {X 0.087,Y -464.203,Z 1067.566,A 0.000,B 0.000,C 90.000,E1 281.895} C_DIS
LIN {X 0.073,Y -468.729,Z 1067.562,A 0.000,B 0.000,C 90.000,E1 281.130} C_DIS
LIN {X 0.089,Y -472.618,Z 1067.558,A 0.000,B 0.000,C 90.000,E1 280.366} C_DIS
LIN {X 0.192,Y -474.868,Z 1067.555,A 0.000,B 0.000,C 90.000,E1 279.849} C_DIS
LIN {X -0.080,Y -476.861,Z 1067.552,A 0.000,B 0.000,C 90.000,E1 279.378} C_DIS
LIN {X 0.048,Y -478.596,Z 1067.549,A 0.000,B 0.000,C 90.000,E1 278.859} C_DIS
LIN {X 0.190,Y -480.121,Z 1067.547,A 0.000,B 0.000,C 90.000,E1 278.341} C_DIS
LIN {X 0.095,Y -482.612,Z 1067.541,A 0.000,B 0.000,C 90.000,E1 277.352} C_DIS
LIN {X -0.214,Y -483.588,Z 1067.538,A 0.000,B 0.000,C 90.000,E1 276.891} C_DIS
LIN {X -0.037,Y -484.342,Z 1067.535,A 0.000,B 0.000,C 90.000,E1 276.372} C_DIS
LIN {X 0.148,Y -484.763,Z 1067.533,A 0.000,B 0.000,C 90.000,E1 275.853} C_DIS
LIN {X -0.148,Y -484.775,Z 1067.530,A 0.000,B 0.000,C 90.000,E1 275.391} C_DIS
LIN {X -0.001,Y -484.379,Z 1067.527,A 0.000,B 0.000,C 90.000,E1 274.878} C_DIS
LIN {X 0.190,Y -483.553,Z 1067.524,A 0.000,B 0.000,C 90.000,E1 274.359} C_DIS
LIN {X -0.108,Y -482.157,Z 1067.522,A 0.000,B 0.000,C 90.000,E1 273.898} C_DIS
LIN {X 0.040,Y -480.173,Z 1067.519,A 0.000,B 0.000,C 90.000,E1 273.383} C_DIS
LIN {X 0.206,Y -477.424,Z 1067.516,A 0.000,B 0.000,C 90.000,E1 272.865} C_DIS
LIN {X 0.030,Y -475.876,Z 1067.515,A 0.000,B 0.000,C 90.000,E1 272.636} C_DIS
LIN {X 0.145,Y -472.008,Z 1067.512,A 0.000,B 0.000,C 90.000,E1 272.121} C_DIS
LIN {X -0.212,Y -467.118,Z 1067.509,A 0.000,B 0.000,C 90.000,E1 271.661} C_DIS
LIN {X 0.051,Y -461.478,Z 1067.506,A 0.000,B 0.000,C 90.000,E1 271.146} C_DIS
LIN {X -0.216,Y -455.419,Z 1067.504,A 0.000,B 0.000,C 90.000,E1 270.745} C_DIS
LIN {X -0.044,Y -448.893,Z 1067.502,A 0.000,B 0.000,C 90.000,E1 270.344} C_DIS
LIN {X 0.130,Y -441.853,Z 1067.500,A 0.000,B 0.000,C 90.000,E1 270.000} C_DIS
LIN {X -0.107,Y -434.281,Z 1067.499,A 0.000,B 0.000,C 90.000,E1 269.771} C_DIS
LIN {X 0.118,Y -426.375,Z 1067.498,A 0.000,B 0.000,C 90.000,E1 269.542} C_DIS
LIN {X -0.089,Y -417.838,Z 1067.497,A 0.000,B 0.000,C 90.000,E1 269.427} C_DIS
LIN {X 0.006,Y -408.867,Z 1067.496,A 0.000,B 0.000,C 90.000,E1 269.312} C_DIS
LIN {X -0.143,Y -396.750,Z 1067.496,A 0.000,B 0.000,C 90.000,E1 269.255} C_DIS
LIN {X 0.191,Y -393.065,Z 1067.496,A 0.000,B 0.000,C 90.000,E1 269.198} C_DIS
LIN {X 0.061,Y -181.369,Z 1067.496,A 0.000,B 0.000,C 90.000,E1 269.198} C_DIS
LIN {X -0.088,Y -180.907,Z 1067.475,A 0.000,B 0.000,C 90.000,E1 265.527} C_DIS
LIN {X -0.031,Y -180.750,Z 1067.470,A 0.000,B 0.000,C 90.000,E1 264.666} C_DIS
LIN {X 0.037,Y -178.841,Z 1067.442,A 0.000,B 0.000,C 90.000,E1 259.577} C_DIS
LIN {X -0.066,Y -175.885,Z 1067.414,A 0.000,B 0.000,C 90.000,E1 254.519} C_DIS
LIN {X 0.040,Y -174.551,Z 1067.404,A 0.000,B 0.000,C 90.000,E1 252.779} C_DIS
LIN {X -0.027,Y -171.535,Z 1067.381,A 0.000,B 0.000,C 90.000,E1 248.518} C_DIS
LIN {X -0.033,Y -167.760,Z 1067.357,A 0.000,B 0.000,C 90.000,E1 244.204} C_DIS
LIN {X -0.091,Y -166.466,Z 1067.347,A 0.000,B 0.000,C 90.000,E1 242.487} C_DIS
LIN {X 0.045,Y -163.181,Z 1067.328,A 0.000,B 0.000,C 90.000,E1 238.948} C_DIS
LIN {X -0.040,Y -161.141,Z 1067.313,A 0.000,B 0.000,C 90.000,E1 236.342} C_DIS
LIN {X -0.003,Y -157.161,Z 1067.288,A 0.000,B 0.000,C 90.000,E1 231.904} C_DIS
LIN {X 0.019,Y -155.893,Z 1067.278,A 0.000,B 0.000,C 90.000,E1 230.114} C_DIS
LIN {X -0.023,Y -152.142,Z 1067.254,A 0.000,B 0.000,C 90.000,E1 225.648} C_DIS
LIN {X -0.003,Y -150.392,Z 1067.239,A 0.000,B 0.000,C 90.000,E1 222.933} C_DIS
LIN {X 0.022,Y -147.123,Z 1067.213,A 0.000,B 0.000,C 90.000,E1 218.382} C_DIS
LIN {X 0.012,Y -145.687,Z 1067.198,A 0.000,B 0.000,C 90.000,E1 215.644} C_DIS
LIN {X 0.010,Y -143.069,Z 1067.172,A 0.000,B 0.000,C 90.000,E1 211.052} C_DIS
LIN {X -0.059,Y -141.689,Z 1067.152,A 0.000,B 0.000,C 90.000,E1 207.385} C_DIS
LIN {X -0.005,Y -139.461,Z 1067.116,A 0.000,B 0.000,C 90.000,E1 200.865} C_DIS
LIN {X -0.035,Y -139.194,Z 1067.106,A 0.000,B 0.000,C 90.000,E1 199.014} C_DIS
LIN {X -0.018,Y -138.325,Z 1067.054,A 0.000,B 0.000,C 90.000,E1 189.670} C_DIS
LIN {X -0.013,Y -139.451,Z 1067.007,A 0.000,B 0.000,C 90.000,E1 181.260} C_DIS
LIN {X 0.067,Y -140.996,Z 1066.976,A 0.000,B 0.000,C 90.000,E1 175.641} C_DIS
LIN {X 0.017,Y -142.750,Z 1066.955,A 0.000,B 0.000,C 90.000,E1 171.951} C_DIS
LIN {X -0.026,Y -145.149,Z 1066.930,A 0.000,B 0.000,C 90.000,E1 167.353} C_DIS
LIN {X -0.034,Y -147.772,Z 1066.909,A 0.000,B 0.000,C 90.000,E1 163.685} C_DIS
LIN {X 0.046,Y -150.448,Z 1066.889,A 0.000,B 0.000,C 90.000,E1 160.007} C_DIS
LIN {X -0.019,Y -153.895,Z 1066.869,A 0.000,B 0.000,C 90.000,E1 156.410} C_DIS
LIN {X -0.026,Y -157.306,Z 1066.849,A 0.000,B 0.000,C 90.000,E1 152.820} C_DIS
LIN {X -0.008,Y -161.491,Z 1066.829,A 0.000,B 0.000,C 90.000,E1 149.253} C_DIS
LIN {X 0.009,Y -165.691,Z 1066.810,A 0.000,B 0.000,C 90.000,E1 145.722} C_DIS
LIN {X -0.104,Y -170.633,Z 1066.790,A 0.000,B 0.000,C 90.000,E1 142.271} C_DIS
LIN {X 0.049,Y -175.509,Z 1066.771,A 0.000,B 0.000,C 90.000,E1 138.771} C_DIS
LIN {X -0.086,Y -181.129,Z 1066.752,A 0.000,B 0.000,C 90.000,E1 135.405} C_DIS
LIN {X 0.041,Y -186.578,Z 1066.733,A 0.000,B 0.000,C 90.000,E1 132.000} C_DIS
LIN {X -0.010,Y -191.191,Z 1066.719,A 0.000,B 0.000,C 90.000,E1 129.519} C_DIS
LIN {X 0.036,Y -196.999,Z 1066.701,A 0.000,B 0.000,C 90.000,E1 126.217} C_DIS
LIN {X 0.073,Y -198.764,Z 1066.696,A 0.000,B 0.000,C 90.000,E1 125.311} C_DIS
LIN {X 0.076,Y -305.542,Z 1066.696,A 0.000,B 0.000,C 90.000,E1 125.311} C_DIS
LIN {X -0.166,Y -307.793,Z 1066.696,A 0.000,B 0.000,C 90.000,E1 125.311} C_DIS
LIN {X -0.030,Y -313.542,Z 1066.694,A 0.000,B 0.000,C 90.000,E1 124.945} C_DIS
LIN {X -0.072,Y -316.605,Z 1066.692,A 0.000,B 0.000,C 90.000,E1 124.612} C_DIS
LIN {X 0.095,Y -318.585,Z 1066.691,A 0.000,B 0.000,C 90.000,E1 124.278} C_DIS
LIN {X 0.000,Y -320.135,Z 1066.689,A 0.000,B 0.000,C 90.000,E1 123.992} C_DIS
LIN {X -0.115,Y -322.514,Z 1066.685,A 0.000,B 0.000,C 90.000,E1 123.372} C_DIS
LIN {X -0.045,Y -332.881,Z 1066.669,A 0.000,B 0.000,C 90.000,E1 120.512} C_DIS
LIN {X -0.063,Y -344.594,Z 1066.654,A 0.000,B 0.000,C 90.000,E1 117.719} C_DIS
LIN {X 0.109,Y -357.750,Z 1066.639,A 0.000,B 0.000,C 90.000,E1 114.951} C_DIS
LIN {X -0.032,Y -370.752,Z 1066.625,A 0.000,B 0.000,C 90.000,E1 112.589} C_DIS
LIN {X 0.016,Y -385.080,Z 1066.613,A 0.000,B 0.000,C 90.000,E1 110.248} C_DIS
LIN {X -0.217,Y -400.834,Z 1066.600,A 0.000,B 0.000,C 90.000,E1 108.000} C_DIS
LIN {X 0.083,Y -418.129,Z 1066.588,A 0.000,B 0.000,C 90.000,E1 105.733} C_DIS
LIN {X -0.100,Y -437.075,Z 1066.575,A 0.000,B 0.000,C 90.000,E1 103.592} C_DIS
LIN {X 0.046,Y -457.116,Z 1066.564,A 0.000,B 0.000,C 90.000,E1 101.535} C_DIS
LIN {X -0.138,Y -467.340,Z 1066.559,A 0.000,B 0.000,C 90.000,E1 100.602} C_DIS
LIN {X -0.122,Y -469.467,Z 1066.557,A 0.000,B 0.000,C 90.000,E1 100.366} C_DIS
LIN {X 0.189,Y -471.199,Z 1066.556,A 0.000,B 0.000,C 90.000,E1 100.074} C_DIS
LIN {X -0.045,Y -472.500,Z 1066.555,A 0.000,B 0.000,C 90.000,E1 99.849} C_DIS
LIN {X 0.138,Y -474.117,Z 1066.552,A 0.000,B 0.000,C 90.000,E1 99.321} C_DIS
LIN {X -0.218,Y -474.678,Z 1066.549,A 0.000,B 0.000,C 90.000,E1 98.859} C_DIS
LIN {X -0.094,Y -474.273,Z 1066.546,A 0.000,B 0.000,C 90.000,E1 98.341} C_DIS
LIN {X 0.101,Y -472.847,Z 1066.543,A 0.000,B 0.000,C 90.000,E1 97.814} C_DIS
LIN {X -0.101,Y -471.678,Z 1066.542,A 0.000,B 0.000,C 90.000,E1 97.587} C_DIS
LIN {X 0.226,Y -470.122,Z 1066.541,A 0.000,B 0.000,C 90.000,E1 97.296} C_DIS
LIN {X 0.082,Y -455.805,Z 1066.529,A 0.000,B 0.000,C 90.000,E1 95.277} C_DIS
LIN {X -0.004,Y -441.607,Z 1066.518,A 0.000,B 0.000,C 90.000,E1 93.212} C_DIS
LIN {X 0.012,Y -423.845,Z 1066.502,A 0.000,B 0.000,C 90.000,E1 90.286} C_DIS
LIN {X -0.115,Y -407.376,Z 1066.485,A 0.000,B 0.000,C 90.000,E1 87.306} C_DIS
LIN {X -0.120,Y -398.418,Z 1066.476,A 0.000,B 0.000,C 90.000,E1 85.641} C_DIS
LIN {X 0.142,Y -389.255,Z 1066.466,A 0.000,B 0.000,C 90.000,E1 83.913} C_DIS
LIN {X -0.128,Y -378.350,Z 1066.455,A 0.000,B 0.000,C 90.000,E1 81.951} C_DIS
LIN {X -0.129,Y -368.727,Z 1066.445,A 0.000,B 0.000,C 90.000,E1 80.208} C_DIS
LIN {X 0.048,Y -358.807,Z 1066.436,A 0.000,B 0.000,C 90.000,E1 78.409} C_DIS
LIN {X 0.108,Y -347.130,Z 1066.424,A 0.000,B 0.000,C 90.000,E1 76.297} C_DIS
LIN {X -0.044,Y -332.430,Z 1066.409,A 0.000,B 0.000,C 90.000,E1 73.559} C_DIS
LIN {X -0.068,Y -318.295,Z 1066.393,A 0.000,B 0.000,C 90.000,E1 70.732} C_DIS
LIN {X 0.025,Y -303.471,Z 1066.375,A 0.000,B 0.000,C 90.000,E1 67.486} C_DIS
LIN {X 0.010,Y -292.072,Z 1066.360,A 0.000,B 0.000,C 90.000,E1 64.845} C_DIS
LIN {X 0.002,Y -282.218,Z 1066.347,A 0.000,B 0.000,C 90.000,E1 62.487} C_DIS
LIN {X -0.024,Y -271.287,Z 1066.332,A 0.000,B 0.000,C 90.000,E1 59.744} C_DIS
LIN {X 0.086,Y -260.590,Z 1066.316,A 0.000,B 0.000,C 90.000,E1 56.914} C_DIS
LIN {X 0.016,Y -249.013,Z 1066.298,A 0.000,B 0.000,C 90.000,E1 53.703} C_DIS
LIN {X -0.127,Y -237.974,Z 1066.280,A 0.000,B 0.000,C 90.000,E1 50.436} C_DIS
LIN {X 0.081,Y -228.822,Z 1066.263,A 0.000,B 0.000,C 90.000,E1 47.391} C_DIS
LIN {X 0.131,Y -219.207,Z 1066.244,A 0.000,B 0.000,C 90.000,E1 43.947} C_DIS
LIN {X 0.047,Y -211.116,Z 1066.227,A 0.000,B 0.000,C 90.000,E1 40.862} C_DIS
LIN {X -0.048,Y -203.503,Z 1066.209,A 0.000,B 0.000,C 90.000,E1 37.729} C_DIS
LIN {X 0.066,Y -196.482,Z 1066.192,A 0.000,B 0.000,C 90.000,E1 34.485} C_DIS
LIN {X -0.052,Y -190.137,Z 1066.174,A 0.000,B 0.000,C 90.000,E1 31.258} C_DIS
LIN {X 0.038,Y -184.505,Z 1066.155,A 0.000,B 0.000,C 90.000,E1 27.924} C_DIS
LIN {X -0.013,Y -179.603,Z 1066.137,A 0.000,B 0.000,C 90.000,E1 24.591} C_DIS
LIN {X -0.080,Y -175.378,Z 1066.118,A 0.000,B 0.000,C 90.000,E1 21.227} C_DIS
LIN {X 0.052,Y -171.907,Z 1066.099,A 0.000,B 0.000,C 90.000,E1 17.764} C_DIS
LIN {X -0.028,Y -168.487,Z 1066.075,A 0.000,B 0.000,C 90.000,E1 13.480} C_DIS
LIN {X -0.060,Y -165.809,Z 1066.046,A 0.000,B 0.000,C 90.000,E1 8.276} C_DIS
LIN {X -0.020,Y -166.342,Z 1065.954,A 0.000,B 0.000,C 90.000,E1 351.659} C_DIS
LIN {X -0.004,Y -168.843,Z 1065.929,A 0.000,B 0.000,C 90.000,E1 347.297} C_DIS
LIN {X 0.023,Y -172.445,Z 1065.905,A 0.000,B 0.000,C 90.000,E1 342.960} C_DIS
LIN {X 0.047,Y -176.026,Z 1065.886,A 0.000,B 0.000,C 90.000,E1 339.518} C_DIS
LIN {X 0.079,Y -180.376,Z 1065.867,A 0.000,B 0.000,C 90.000,E1 336.102} C_DIS
LIN {X 0.041,Y -185.408,Z 1065.849,A 0.000,B 0.000,C 90.000,E1 332.743} C_DIS
LIN {X 0.048,Y -191.303,Z 1065.830,A 0.000,B 0.000,C 90.000,E1 329.410} C_DIS
LIN {X 0.006,Y -198.011,Z 1065.812,A 0.000,B 0.000,C 90.000,E1 326.135} C_DIS
LIN {X -0.089,Y -205.413,Z 1065.794,A 0.000,B 0.000,C 90.000,E1 322.924} C_DIS
LIN {X 0.102,Y -214.617,Z 1065.774,A 0.000,B 0.000,C 90.000,E1 319.299} C_DIS
LIN {X -0.015,Y -223.477,Z 1065.757,A 0.000,B 0.000,C 90.000,E1 316.215} C_DIS
LIN {X -0.032,Y -231.919,Z 1065.742,A 0.000,B 0.000,C 90.000,E1 313.542} C_DIS
LIN {X -0.028,Y -242.893,Z 1065.725,A 0.000,B 0.000,C 90.000,E1 310.539} C_DIS
LIN {X 0.099,Y -250.633,Z 1065.715,A 0.000,B 0.000,C 90.000,E1 308.669} C_DIS
LIN {X 0.073,Y -261.054,Z 1065.703,A 0.000,B 0.000,C 90.000,E1 306.503} C_DIS
LIN {X -0.133,Y -278.429,Z 1065.685,A 0.000,B 0.000,C 90.000,E1 303.372} C_DIS
LIN {X 0.103,Y -297.183,Z 1065.668,A 0.000,B 0.000,C 90.000,E1 300.256} C_DIS
LIN {X -0.024,Y -315.051,Z 1065.654,A 0.000,B 0.000,C 90.000,E1 297.641} C_DIS
LIN {X -0.044,Y -329.444,Z 1065.643,A 0.000,B 0.000,C 90.000,E1 295.720} C_DIS
LIN {X -0.016,Y -339.834,Z 1065.636,A 0.000,B 0.000,C 90.000,E1 294.463} C_DIS
LIN {X 0.003,Y -353.173,Z 1065.628,A 0.000,B 0.000,C 90.000,E1 293.025} C_DIS
LIN {X -0.145,Y -372.078,Z 1065.618,A 0.000,B 0.000,C 90.000,E1 291.227} C_DIS
LIN {X -0.009,Y -391.332,Z 1065.608,A 0.000,B 0.000,C 90.000,E1 289.504} C_DIS
LIN {X 0.052,Y -405.157,Z 1065.602,A 0.000,B 0.000,C 90.000,E1 288.308} C_DIS
LIN {X 0.125,Y -415.893,Z 1065.596,A 0.000,B 0.000,C 90.000,E1 287.347} C_DIS
LIN {X 0.006,Y -426.272,Z 1065.591,A 0.000,B 0.000,C 90.000,E1 286.386} C_DIS
LIN {X 0.164,Y -433.742,Z 1065.587,A 0.000,B 0.000,C 90.000,E1 285.607} C_DIS
LIN {X -0.134,Y -443.424,Z 1065.581,A 0.000,B 0.000,C 90.000,E1 284.592} C_DIS
LIN {X -0.099,Y -452.392,Z 1065.575,A 0.000,B 0.000,C 90.000,E1 283.536} C_DIS
LIN {X -0.217,Y -458.423,Z 1065.571,A 0.000,B 0.000,C 90.000,E1 282.771} C_DIS
LIN {X 0.164,Y -463.761,Z 1065.567,A 0.000,B 0.000,C 90.000,E1 281.951} C_DIS
LIN {X -0.160,Y -466.969,Z 1065.564,A 0.000,B 0.000,C 90.000,E1 281.478} C_DIS
LIN {X -0.157,Y -471.134,Z 1065.559,A 0.000,B 0.000,C 90.000,E1 280.715} C_DIS
LIN {X -0.209,Y -474.647,Z 1065.555,A 0.000,B 0.000,C 90.000,E1 279.962} C_DIS
LIN {X -0.092,Y -476.708,Z 1065.552,A 0.000,B 0.000,C 90.000,E1 279.443} C_DIS
LIN {X 0.117,Y -478.494,Z 1065.550,A 0.000,B 0.000,C 90.000,E1 278.916} C_DIS
LIN {X -0.217,Y -480.069,Z 1065.547,A 0.000,B 0.000,C 90.000,E1 278.454} C_DIS
LIN {X 0.162,Y -482.612,Z 1065.541,A 0.000,B 0.000,C 90.000,E1 277.409} C_DIS
LIN {X -0.147,Y -483.649,Z 1065.538,A 0.000,B 0.000,C 90.000,E1 276.947} C_DIS
LIN {X 0.030,Y -484.463,Z 1065.536,A 0.000,B 0.000,C 90.000,E1 276.429} C_DIS
LIN {X 0.213,Y -484.968,Z 1065.533,A 0.000,B 0.000,C 90.000,E1 275.910} C_DIS
LIN {X -0.127,Y -485.004,Z 1065.530,A 0.000,B 0.000,C 90.000,E1 275.454} C_DIS
LIN {X 0.066,Y -484.702,Z 1065.527,A 0.000,B 0.000,C 90.000,E1 274.935} C_DIS
LIN {X -0.226,Y -483.935,Z 1065.525,A 0.000,B 0.000,C 90.000,E1 274.473} C_DIS
LIN {X -0.039,Y -482.615,Z 1065.522,A 0.000,B 0.000,C 90.000,E1 273.955} C_DIS
LIN {X 0.110,Y -480.706,Z 1065.519,A 0.000,B 0.000,C 90.000,E1 273.440} C_DIS
LIN {X -0.198,Y -478.139,Z 1065.516,A 0.000,B 0.000,C 90.000,E1 272.980} C_DIS
LIN {X -0.070,Y -474.787,Z 1065.514,A 0.000,B 0.000,C 90.000,E1 272.465} C_DIS
LIN {X 0.223,Y -472.830,Z 1065.512,A 0.000,B 0.000,C 90.000,E1 272.178} C_DIS
LIN {X -0.132,Y -468.076,Z 1065.509,A 0.000,B 0.000,C 90.000,E1 271.718} C_DIS
LIN {X 0.103,Y -462.552,Z 1065.507,A 0.000,B 0.000,C 90.000,E1 271.203} C_DIS
LIN {X 0.220,Y -456.582,Z 1065.504,A 0.000,B 0.000,C 90.000,E1 270.745} C_DIS
LIN {X -0.145,Y -450.136,Z 1065.502,A 0.000,B 0.000,C 90.000,E1 270.401} C_DIS
LIN {X -0.043,Y -443.219,Z 1065.500,A 0.000,B 0.000,C 90.000,E1 270.057} C_DIS
LIN {X 0.103,Y -435.919,Z 1065.499,A 0.000,B 0.000,C 90.000,E1 269.771} C_DIS
LIN {X -0.150,Y -428.081,Z 1065.498,A 0.000,B 0.000,C 90.000,E1 269.599} C_DIS
LIN {X -0.015,Y -419.786,Z 1065.497,A 0.000,B 0.000,C 90.000,E1 269.427} C_DIS
LIN {X 0.014,Y -410.551,Z 1065.496,A 0.000,B 0.000,C 90.000,E1 269.312} C_DIS
LIN {X -0.160,Y -399.632,Z 1065.496,A 0.000,B 0.000,C 90.000,E1 269.255} C_DIS
LIN {X 0.108,Y -394.299,Z 1065.496,A 0.000,B 0.000,C 90.000,E1 269.198} C_DIS
LIN {X 0.020,Y -181.365,Z 1065.496,A 0.000,B 0.000,C 90.000,E1 269.198} C_DIS
LIN {X 0.077,Y -180.907,Z 1065.475,A 0.000,B 0.000,C 90.000,E1 265.469} C_DIS
LIN {X -0.046,Y -180.747,Z 1065.470,A 0.000,B 0.000,C 90.000,E1 264.666} C_DIS
LIN {X 0.023,Y -178.839,Z 1065.442,A 0.000,B 0.000,C 90.000,E1 259.577} C_DIS
LIN {X -0.081,Y -175.883,Z 1065.414,A 0.000,B 0.000,C 90.000,E1 254.519} C_DIS
LIN {X 0.025,Y -174.547,Z 1065.404,A 0.000,B 0.000,C 90.000,E1 252.779} C_DIS
LIN {X -0.043,Y -171.531,Z 1065.381,A 0.000,B 0.000,C 90.000,E1 248.518} C_DIS
LIN {X -0.049,Y -167.756,Z 1065.357,A 0.000,B 0.000,C 90.000,E1 244.204} C_DIS
LIN {X 0.042,Y -166.462,Z 1065.347,A 0.000,B 0.000,C 90.000,E1 242.436} C_DIS
LIN {X 0.031,Y -163.177,Z 1065.328,A 0.000,B 0.000,C 90.000,E1 238.948} C_DIS
LIN {X 0.080,Y -161.136,Z 1065.313,A 0.000,B 0.000,C 90.000,E1 236.294} C_DIS
LIN {X -0.018,Y -157.157,Z 1065.288,A 0.000,B 0.000,C 90.000,E1 231.904} C_DIS
LIN {X 0.006,Y -155.889,Z 1065.278,A 0.000,B 0.000,C 90.000,E1 230.114} C_DIS
LIN {X -0.036,Y -152.138,Z 1065.254,A 0.000,B 0.000,C 90.000,E1 225.648} C_DIS
LIN {X -0.017,Y -150.389,Z 1065.239,A 0.000,B 0.000,C 90.000,E1 222.933} C_DIS
LIN {X 0.008,Y -147.120,Z 1065.213,A 0.000,B 0.000,C 90.000,E1 218.382} C_DIS
LIN {X -0.001,Y -145.685,Z 1065.198,A 0.000,B 0.000,C 90.000,E1 215.644} C_DIS
LIN {X -0.004,Y -143.067,Z 1065.172,A 0.000,B 0.000,C 90.000,E1 211.052} C_DIS
LIN {X -0.072,Y -141.688,Z 1065.152,A 0.000,B 0.000,C 90.000,E1 207.385} C_DIS
LIN {X -0.017,Y -139.460,Z 1065.116,A 0.000,B 0.000,C 90.000,E1 200.865} C_DIS
LIN {X 0.083,Y -139.194,Z 1065.105,A 0.000,B 0.000,C 90.000,E1 198.960} C_DIS
LIN {X -0.031,Y -138.325,Z 1065.054,A 0.000,B 0.000,C 90.000,E1 189.670} C_DIS
LIN {X -0.026,Y -139.452,Z 1065.007,A 0.000,B 0.000,C 90.000,E1 181.260} C_DIS
LIN {X 0.054,Y -140.998,Z 1064.976,A 0.000,B 0.000,C 90.000,E1 175.641} C_DIS
LIN {X 0.004,Y -142.753,Z 1064.955,A 0.000,B 0.000,C 90.000,E1 171.951} C_DIS
LIN {X -0.040,Y -145.152,Z 1064.930,A 0.000,B 0.000,C 90.000,E1 167.353} C_DIS
LIN {X -0.046,Y -147.776,Z 1064.909,A 0.000,B 0.000,C 90.000,E1 163.685} C_DIS
LIN {X 0.032,Y -150.452,Z 1064.889,A 0.000,B 0.000,C 90.000,E1 160.007} C_DIS
LIN {X -0.034,Y -153.900,Z 1064.869,A 0.000,B 0.000,C 90.000,E1 156.410} C_DIS
LIN {X 0.031,Y -157.311,Z 1064.849,A 0.000,B 0.000,C 90.000,E1 152.794} C_DIS
LIN {X -0.021,Y -161.498,Z 1064.829,A 0.000,B 0.000,C 90.000,E1 149.253} C_DIS
LIN {X -0.006,Y -165.697,Z 1064.810,A 0.000,B 0.000,C 90.000,E1 145.722} C_DIS
LIN {X -0.015,Y -170.641,Z 1064.790,A 0.000,B 0.000,C 90.000,E1 142.236} C_DIS
LIN {X 0.033,Y -175.517,Z 1064.771,A 0.000,B 0.000,C 90.000,E1 138.771} C_DIS
LIN {X -0.101,Y -181.137,Z 1064.752,A 0.000,B 0.000,C 90.000,E1 135.405} C_DIS
LIN {X 0.026,Y -186.587,Z 1064.733,A 0.000,B 0.000,C 90.000,E1 132.000} C_DIS
LIN {X -0.025,Y -191.199,Z 1064.719,A 0.000,B 0.000,C 90.000,E1 129.519} C_DIS
LIN {X 0.021,Y -197.009,Z 1064.701,A 0.000,B 0.000,C 90.000,E1 126.217} C_DIS
LIN {X -0.037,Y -198.666,Z 1064.697,A 0.000,B 0.000,C 90.000,E1 125.391} C_DIS
LIN {X -0.109,Y -305.281,Z 1064.697,A 0.000,B 0.000,C 90.000,E1 125.391} C_DIS
LIN {X 0.158,Y -307.043,Z 1064.696,A 0.000,B 0.000,C 90.000,E1 125.311} C_DIS
LIN {X 0.014,Y -311.188,Z 1064.695,A 0.000,B 0.000,C 90.000,E1 125.152} C_DIS
LIN {X -0.057,Y -313.551,Z 1064.694,A 0.000,B 0.000,C 90.000,E1 124.978} C_DIS
LIN {X -0.097,Y -316.790,Z 1064.692,A 0.000,B 0.000,C 90.000,E1 124.612} C_DIS
LIN {X 0.025,Y -318.732,Z 1064.690,A 0.000,B 0.000,C 90.000,E1 124.278} C_DIS
LIN {X -0.115,Y -320.251,Z 1064.689,A 0.000,B 0.000,C 90.000,E1 123.992} C_DIS
LIN {X 0.033,Y -323.650,Z 1064.683,A 0.000,B 0.000,C 90.000,E1 123.007} C_DIS
LIN {X -0.043,Y -334.173,Z 1064.668,A 0.000,B 0.000,C 90.000,E1 120.178} C_DIS
LIN {X -0.021,Y -346.048,Z 1064.652,A 0.000,B 0.000,C 90.000,E1 117.385} C_DIS
LIN {X 0.032,Y -359.385,Z 1064.637,A 0.000,B 0.000,C 90.000,E1 114.643} C_DIS
LIN {X -0.068,Y -372.559,Z 1064.624,A 0.000,B 0.000,C 90.000,E1 112.280} C_DIS
LIN {X 0.026,Y -387.070,Z 1064.611,A 0.000,B 0.000,C 90.000,E1 109.939} C_DIS
LIN {X -0.163,Y -403.024,Z 1064.598,A 0.000,B 0.000,C 90.000,E1 107.692} C_DIS
LIN {X 0.188,Y -420.532,Z 1064.586,A 0.000,B 0.000,C 90.000,E1 105.426} C_DIS
